KUKA KRL program: NEW_MASTER_MESA_A.src, NEW_MASTER_MESA_A.dat

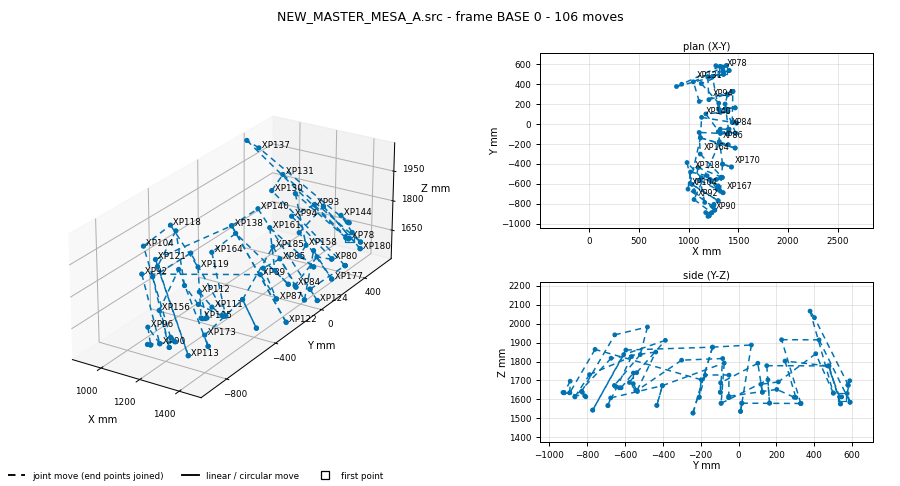
[picture p0: tool path of NEW_MASTER_MESA_A.src in frame BASE 0, 106 of 108 moves have a stored position in this frame; points joined in program order, loops and branches not executed]
--- NEW_MASTER_MESA_A.src ---
&ACCESS RVP
&REL 381
&PARAM EDITMASK = *
&PARAM TEMPLATE = C:\KRC\Roboter\Template\vorgabe
&PARAM DISKPATH = KRC:\R1\Program\Solda\MASTER_125
DEF NEW_MASTER_MESA_A( )
;FOLD INI;%{PE}
  ;FOLD BASISTECH INI
    GLOBAL INTERRUPT DECL 3 WHEN $STOPMESS==TRUE DO IR_STOPM ( )
    INTERRUPT ON 3
    BAS (#INITMOV,0 )
  ;ENDFOLD (BASISTECH INI)
  ;FOLD USER INI
    ;Make your modifications here

  ;ENDFOLD (USER INI)
;ENDFOLD (INI)

;FOLD PTP HOME  Vel= 100 % DEFAULT;%{PE}%MKUKATPBASIS,%CMOVE,%VPTP,%P 1:PTP, 2:HOME, 3:, 5:100, 7:DEFAULT
$BWDSTART = FALSE
PDAT_ACT=PDEFAULT
FDAT_ACT=FHOME
BAS (#PTP_PARAMS,100 )
$H_POS=XHOME
PTP  XHOME
;ENDFOLD
;FOLD ; CORDAO 01;%{PE}%R 8.3.48,%MKUKATPBASIS,%CCOMMENT,%VNORMAL,%P 2:CORDAO 01
;ENDFOLD
;FOLD ARCON WDAT39 PTP P78 Vel=100 % PDAT60 Tool[1]:TOCH Base[0] ;%{PE}
;FOLD Parameters ;%{h}
;Params IlfProvider=kukaroboter.arctech.arconptp; Kuka.PointName=P78; Kuka.BlendingEnabled=False; Kuka.MoveDataPtpName=PDAT60; Kuka.VelocityPtp=100; Kuka.MovementParameterFieldEnabled=True; ArcTech.WdatVarName=WDAT39; ArcTech.SeamName=
;ENDFOLD
$BWDSTART = FALSE
PDAT_ACT = PPDAT60
FDAT_ACT = FP78
BAS(#PTP_PARAMS, 100.0)
TRIGGER WHEN DISTANCE = 1 DELAY = ATBg_PreDefinitionTime DO Arc_DefineStrikeParams(3, AS_WDAT39) PRIO = -1
Arc_DefineCpPattern(#OffInAdvance, WV_WDAT39, TRUE)
PTP XP78
Arc_On(3, AS_WDAT39, ATBg_StartErrSetField[1], AW_WDAT39, WV_WDAT39, ATBg_WeldErrSetField[1], #StdArcOn, " ")
Arc_DefineCpPattern(#OnInAdvance, WV_WDAT39, TRUE)
;ENDFOLD
;FOLD ARCOFF WDAT40 LIN P79 CPDAT22 Tool[1]:TOCH Base[0] ;%{PE}
;FOLD Parameters ;%{h}
;Params IlfProvider=kukaroboter.arctech.arcofflin; Kuka.PointName=P79; Kuka.BlendingEnabled=False; Kuka.MoveDataName=CPDAT22;  Kuka.MovementParameterFieldEnabled=True; ArcTech.WdatVarName=WDAT40
;ENDFOLD
$BWDSTART = FALSE
LDAT_ACT = LCPDAT22
FDAT_ACT = FP79
BAS(#CP_PARAMS, ATBg_BAS_VELDefinition)
LIN XP79
Arc_Off(1, AC_WDAT40)
;ENDFOLD
;FOLD PTP P93 CONT Vel=100 % PDAT70 Tool[1]:TOCH Base[0];%{PE}%R 8.3.48,%MKUKATPBASIS,%CMOVE,%VPTP,%P 1:PTP, 2:P93, 3:C_DIS, 5:100, 7:PDAT70
$BWDSTART=FALSE
PDAT_ACT=PPDAT70
FDAT_ACT=FP93
BAS(#PTP_PARAMS,100)
PTP XP93 C_DIS
;ENDFOLD
;FOLD PTP P94 CONT Vel=100 % PDAT71 Tool[1]:TOCH Base[0];%{PE}%R 8.3.48,%MKUKATPBASIS,%CMOVE,%VPTP,%P 1:PTP, 2:P94, 3:C_DIS, 5:100, 7:PDAT71
$BWDSTART=FALSE
PDAT_ACT=PPDAT71
FDAT_ACT=FP94
BAS(#PTP_PARAMS,100)
PTP XP94 C_DIS
;ENDFOLD
;FOLD ; CORDAO 02;%{PE}%R 8.3.48,%MKUKATPBASIS,%CCOMMENT,%VNORMAL,%P 2:CORDAO 02
;ENDFOLD
;FOLD ARCON WDAT41 PTP P80 Vel=100 % PDAT61 Tool[1]:TOCH Base[0] ;%{PE}
;FOLD Parameters ;%{h}
;Params IlfProvider=kukaroboter.arctech.arconptp; Kuka.PointName=P80; Kuka.BlendingEnabled=False; Kuka.MoveDataPtpName=PDAT61; Kuka.VelocityPtp=100; Kuka.MovementParameterFieldEnabled=True; ArcTech.WdatVarName=WDAT41; ArcTech.SeamName=
;ENDFOLD
$BWDSTART = FALSE
PDAT_ACT = PPDAT61
FDAT_ACT = FP80
BAS(#PTP_PARAMS, 100.0)
TRIGGER WHEN DISTANCE = 1 DELAY = ATBg_PreDefinitionTime DO Arc_DefineStrikeParams(1, AS_WDAT41) PRIO = -1
Arc_DefineCpPattern(#OffInAdvance, WV_WDAT41, TRUE)
PTP XP80
Arc_On(1, AS_WDAT41, ATBg_StartErrSetField[1], AW_WDAT41, WV_WDAT41, ATBg_WeldErrSetField[1], #StdArcOn, " ")
Arc_DefineCpPattern(#OnInAdvance, WV_WDAT41, TRUE)
;ENDFOLD
;FOLD ARCOFF WDAT42 LIN P81 CPDAT23 Tool[1]:TOCH Base[0] ;%{PE}
;FOLD Parameters ;%{h}
;Params IlfProvider=kukaroboter.arctech.arcofflin; Kuka.PointName=P81; Kuka.BlendingEnabled=False; Kuka.MoveDataName=CPDAT23;  Kuka.MovementParameterFieldEnabled=True; ArcTech.WdatVarName=WDAT42
;ENDFOLD
$BWDSTART = FALSE
LDAT_ACT = LCPDAT23
FDAT_ACT = FP81
BAS(#CP_PARAMS, ATBg_BAS_VELDefinition)
LIN XP81
Arc_Off(1, AC_WDAT42)
;ENDFOLD
;FOLD PTP P95 CONT Vel=100 % PDAT72 Tool[1]:TOCH Base[0];%{PE}%R 8.3.48,%MKUKATPBASIS,%CMOVE,%VPTP,%P 1:PTP, 2:P95, 3:C_DIS, 5:100, 7:PDAT72
$BWDSTART=FALSE
PDAT_ACT=PPDAT72
FDAT_ACT=FP95
BAS(#PTP_PARAMS,100)
PTP XP95 C_DIS
;ENDFOLD
;FOLD PTP P84 CONT Vel=100 % PDAT63 Tool[1]:TOCH Base[0];%{PE}%R 8.3.48,%MKUKATPBASIS,%CMOVE,%VPTP,%P 1:PTP, 2:P84, 3:C_DIS, 5:100, 7:PDAT63
$BWDSTART=FALSE
PDAT_ACT=PPDAT63
FDAT_ACT=FP84
BAS(#PTP_PARAMS,100)
PTP XP84 C_DIS
;ENDFOLD
;FOLD ; CORDAO 03;%{PE}%R 8.3.48,%MKUKATPBASIS,%CCOMMENT,%VNORMAL,%P 2:CORDAO 03
;ENDFOLD
;FOLD ARCON WDAT43 PTP P82 Vel=100 % PDAT62 Tool[1]:TOCH Base[0] ;%{PE}
;FOLD Parameters ;%{h}
;Params IlfProvider=kukaroboter.arctech.arconptp; Kuka.PointName=P82; Kuka.BlendingEnabled=False; Kuka.MoveDataPtpName=PDAT62; Kuka.VelocityPtp=100; Kuka.MovementParameterFieldEnabled=True; ArcTech.WdatVarName=WDAT43; ArcTech.SeamName=
;ENDFOLD
$BWDSTART = FALSE
PDAT_ACT = PPDAT62
FDAT_ACT = FP82
BAS(#PTP_PARAMS, 100.0)
TRIGGER WHEN DISTANCE = 1 DELAY = ATBg_PreDefinitionTime DO Arc_DefineStrikeParams(1, AS_WDAT43) PRIO = -1
Arc_DefineCpPattern(#OffInAdvance, WV_WDAT43, TRUE)
PTP XP82
Arc_On(1, AS_WDAT43, ATBg_StartErrSetField[1], AW_WDAT43, WV_WDAT43, ATBg_WeldErrSetField[1], #StdArcOn, " ")
Arc_DefineCpPattern(#OnInAdvance, WV_WDAT43, TRUE)
;ENDFOLD
;FOLD ARCOFF WDAT44 LIN P83 CPDAT24 Tool[1]:TOCH Base[0] ;%{PE}
;FOLD Parameters ;%{h}
;Params IlfProvider=kukaroboter.arctech.arcofflin; Kuka.PointName=P83; Kuka.BlendingEnabled=False; Kuka.MoveDataName=CPDAT24;  Kuka.MovementParameterFieldEnabled=True; ArcTech.WdatVarName=WDAT44
;ENDFOLD
$BWDSTART = FALSE
LDAT_ACT = LCPDAT24
FDAT_ACT = FP83
BAS(#CP_PARAMS, ATBg_BAS_VELDefinition)
LIN XP83
Arc_Off(1, AC_WDAT44)
;ENDFOLD
;FOLD PTP P85 CONT Vel=100 % PDAT64 Tool[1]:TOCH Base[0];%{PE}%R 8.3.48,%MKUKATPBASIS,%CMOVE,%VPTP,%P 1:PTP, 2:P85, 3:C_DIS, 5:100, 7:PDAT64
$BWDSTART=FALSE
PDAT_ACT=PPDAT64
FDAT_ACT=FP85
BAS(#PTP_PARAMS,100)
PTP XP85 C_DIS
;ENDFOLD
;FOLD PTP P86 CONT Vel=100 % PDAT65 Tool[1]:TOCH Base[0];%{PE}%R 8.3.48,%MKUKATPBASIS,%CMOVE,%VPTP,%P 1:PTP, 2:P86, 3:C_DIS, 5:100, 7:PDAT65
$BWDSTART=FALSE
PDAT_ACT=PPDAT65
FDAT_ACT=FP86
BAS(#PTP_PARAMS,100)
PTP XP86 C_DIS
;ENDFOLD
;FOLD ; CORDAO 04;%{PE}%R 8.3.48,%MKUKATPBASIS,%CCOMMENT,%VNORMAL,%P 2:CORDAO 04
;ENDFOLD
;FOLD ARCON WDAT45 PTP P87 Vel=100 % PDAT66 Tool[1]:TOCH Base[0] ;%{PE}
;FOLD Parameters ;%{h}
;Params IlfProvider=kukaroboter.arctech.arconptp; Kuka.PointName=P87; Kuka.BlendingEnabled=False; Kuka.MoveDataPtpName=PDAT66; Kuka.VelocityPtp=100; Kuka.MovementParameterFieldEnabled=True; ArcTech.WdatVarName=WDAT45; ArcTech.SeamName=
;ENDFOLD
$BWDSTART = FALSE
PDAT_ACT = PPDAT66
FDAT_ACT = FP87
BAS(#PTP_PARAMS, 100.0)
TRIGGER WHEN DISTANCE = 1 DELAY = ATBg_PreDefinitionTime DO Arc_DefineStrikeParams(1, AS_WDAT45) PRIO = -1
Arc_DefineCpPattern(#OffInAdvance, WV_WDAT45, TRUE)
PTP XP87
Arc_On(1, AS_WDAT45, ATBg_StartErrSetField[1], AW_WDAT45, WV_WDAT45, ATBg_WeldErrSetField[1], #StdArcOn, " ")
Arc_DefineCpPattern(#OnInAdvance, WV_WDAT45, TRUE)
;ENDFOLD
;FOLD ARCOFF WDAT46 LIN P88 CPDAT25 Tool[1]:TOCH Base[0] ;%{PE}
;FOLD Parameters ;%{h}
;Params IlfProvider=kukaroboter.arctech.arcofflin; Kuka.PointName=P88; Kuka.BlendingEnabled=False; Kuka.MoveDataName=CPDAT25;  Kuka.MovementParameterFieldEnabled=True; ArcTech.WdatVarName=WDAT46
;ENDFOLD
$BWDSTART = FALSE
LDAT_ACT = LCPDAT25
FDAT_ACT = FP88
BAS(#CP_PARAMS, ATBg_BAS_VELDefinition)
LIN XP88
Arc_Off(1, AC_WDAT46)
;ENDFOLD
;FOLD PTP P89 CONT Vel=100 % PDAT67 Tool[1]:TOCH Base[0];%{PE}%R 8.3.48,%MKUKATPBASIS,%CMOVE,%VPTP,%P 1:PTP, 2:P89, 3:C_DIS, 5:100, 7:PDAT67
$BWDSTART=FALSE
PDAT_ACT=PPDAT67
FDAT_ACT=FP89
BAS(#PTP_PARAMS,100)
PTP XP89 C_DIS
;ENDFOLD
;FOLD PTP P92 CONT Vel=100 % PDAT69 Tool[1]:TOCH Base[0];%{PE}%R 8.3.48,%MKUKATPBASIS,%CMOVE,%VPTP,%P 1:PTP, 2:P92, 3:C_DIS, 5:100, 7:PDAT69
$BWDSTART=FALSE
PDAT_ACT=PPDAT69
FDAT_ACT=FP92
BAS(#PTP_PARAMS,100)
PTP XP92 C_DIS
;ENDFOLD
;FOLD ; CORDAO 05;%{PE}%R 8.3.48,%MKUKATPBASIS,%CCOMMENT,%VNORMAL,%P 2:CORDAO 05
;ENDFOLD
;FOLD ARCON WDAT47 PTP P90 Vel=100 % PDAT68 Tool[1]:TOCH Base[0] ;%{PE}
;FOLD Parameters ;%{h}
;Params IlfProvider=kukaroboter.arctech.arconptp; Kuka.PointName=P90; Kuka.BlendingEnabled=False; Kuka.MoveDataPtpName=PDAT68; Kuka.VelocityPtp=100; Kuka.MovementParameterFieldEnabled=True; ArcTech.WdatVarName=WDAT47; ArcTech.SeamName=
;ENDFOLD
$BWDSTART = FALSE
PDAT_ACT = PPDAT68
FDAT_ACT = FP90
BAS(#PTP_PARAMS, 100.0)
TRIGGER WHEN DISTANCE = 1 DELAY = ATBg_PreDefinitionTime DO Arc_DefineStrikeParams(1, AS_WDAT47) PRIO = -1
Arc_DefineCpPattern(#OffInAdvance, WV_WDAT47, TRUE)
PTP XP90
Arc_On(1, AS_WDAT47, ATBg_StartErrSetField[1], AW_WDAT47, WV_WDAT47, ATBg_WeldErrSetField[1], #StdArcOn, " ")
Arc_DefineCpPattern(#OnInAdvance, WV_WDAT47, TRUE)
;ENDFOLD
;FOLD ARCOFF WDAT48 LIN P91 CPDAT26 Tool[1]:TOCH Base[0] ;%{PE}
;FOLD Parameters ;%{h}
;Params IlfProvider=kukaroboter.arctech.arcofflin; Kuka.PointName=P91; Kuka.BlendingEnabled=False; Kuka.MoveDataName=CPDAT26;  Kuka.MovementParameterFieldEnabled=True; ArcTech.WdatVarName=WDAT48
;ENDFOLD
$BWDSTART = FALSE
LDAT_ACT = LCPDAT26
FDAT_ACT = FP91
BAS(#CP_PARAMS, ATBg_BAS_VELDefinition)
LIN XP91
Arc_Off(1, AC_WDAT48)
;ENDFOLD
;FOLD PTP P96 CONT Vel=100 % PDAT73 Tool[1]:TOCH Base[0];%{PE}%R 8.3.48,%MKUKATPBASIS,%CMOVE,%VPTP,%P 1:PTP, 2:P96, 3:C_DIS, 5:100, 7:PDAT73
$BWDSTART=FALSE
PDAT_ACT=PPDAT73
FDAT_ACT=FP96
BAS(#PTP_PARAMS,100)
PTP XP96 C_DIS
;ENDFOLD
;FOLD ; CORDAO 06;%{PE}%R 8.3.48,%MKUKATPBASIS,%CCOMMENT,%VNORMAL,%P 2:CORDAO 06
;ENDFOLD
;FOLD ARCON WDAT49 PTP P97 Vel=100 % PDAT74 Tool[1]:TOCH Base[0] ;%{PE}
;FOLD Parameters ;%{h}
;Params IlfProvider=kukaroboter.arctech.arconptp; Kuka.PointName=P97; Kuka.BlendingEnabled=False; Kuka.MoveDataPtpName=PDAT74; Kuka.VelocityPtp=100; Kuka.MovementParameterFieldEnabled=True; ArcTech.WdatVarName=WDAT49; ArcTech.SeamName=
;ENDFOLD
$BWDSTART = FALSE
PDAT_ACT = PPDAT74
FDAT_ACT = FP97
BAS(#PTP_PARAMS, 100.0)
TRIGGER WHEN DISTANCE = 1 DELAY = ATBg_PreDefinitionTime DO Arc_DefineStrikeParams(1, AS_WDAT49) PRIO = -1
Arc_DefineCpPattern(#OffInAdvance, WV_WDAT49, TRUE)
PTP XP97
Arc_On(1, AS_WDAT49, ATBg_StartErrSetField[1], AW_WDAT49, WV_WDAT49, ATBg_WeldErrSetField[1], #StdArcOn, " ")
Arc_DefineCpPattern(#OnInAdvance, WV_WDAT49, TRUE)
;ENDFOLD
;FOLD ARCOFF WDAT50 LIN P98 CPDAT27 Tool[1]:TOCH Base[0] ;%{PE}
;FOLD Parameters ;%{h}
;Params IlfProvider=kukaroboter.arctech.arcofflin; Kuka.PointName=P98; Kuka.BlendingEnabled=False; Kuka.MoveDataName=CPDAT27;  Kuka.MovementParameterFieldEnabled=True; ArcTech.WdatVarName=WDAT50
;ENDFOLD
$BWDSTART = FALSE
LDAT_ACT = LCPDAT27
FDAT_ACT = FP98
BAS(#CP_PARAMS, ATBg_BAS_VELDefinition)
LIN XP98
Arc_Off(1, AC_WDAT50)
;ENDFOLD
;FOLD ARCOFF WDAT51 LIN P99 CPDAT28 Tool[1]:TOCH Base[0] ;%{PE}
;FOLD Parameters ;%{h}
;Params IlfProvider=kukaroboter.arctech.arcofflin; Kuka.PointName=P99; Kuka.BlendingEnabled=False; Kuka.MoveDataName=CPDAT28;  Kuka.MovementParameterFieldEnabled=True; ArcTech.WdatVarName=WDAT51
;ENDFOLD
$BWDSTART = FALSE
LDAT_ACT = LCPDAT28
FDAT_ACT = FP99
BAS(#CP_PARAMS, ATBg_BAS_VELDefinition)
LIN XP99
Arc_Off(1, AC_WDAT51)
;ENDFOLD
;FOLD ; CORDAO 07;%{PE}%R 8.3.48,%MKUKATPBASIS,%CCOMMENT,%VNORMAL,%P 2:CORDAO 07
;ENDFOLD
;FOLD ARCON WDAT52 PTP P100 Vel=100 % PDAT75 Tool[1]:TOCH Base[0] ;%{PE}
;FOLD Parameters ;%{h}
;Params IlfProvider=kukaroboter.arctech.arconptp; Kuka.PointName=P100; Kuka.BlendingEnabled=False; Kuka.MoveDataPtpName=PDAT75; Kuka.VelocityPtp=100; Kuka.MovementParameterFieldEnabled=True; ArcTech.WdatVarName=WDAT52; ArcTech.SeamName=
;ENDFOLD
$BWDSTART = FALSE
PDAT_ACT = PPDAT75
FDAT_ACT = FP100
BAS(#PTP_PARAMS, 100.0)
TRIGGER WHEN DISTANCE = 1 DELAY = ATBg_PreDefinitionTime DO Arc_DefineStrikeParams(1, AS_WDAT52) PRIO = -1
Arc_DefineCpPattern(#OffInAdvance, WV_WDAT52, TRUE)
PTP XP100
Arc_On(1, AS_WDAT52, ATBg_StartErrSetField[1], AW_WDAT52, WV_WDAT52, ATBg_WeldErrSetField[1], #StdArcOn, " ")
Arc_DefineCpPattern(#OnInAdvance, WV_WDAT52, TRUE)
;ENDFOLD
;FOLD ARCOFF WDAT53 LIN P101 CPDAT29 Tool[1]:TOCH Base[0] ;%{PE}
;FOLD Parameters ;%{h}
;Params IlfProvider=kukaroboter.arctech.arcofflin; Kuka.PointName=P101; Kuka.BlendingEnabled=False; Kuka.MoveDataName=CPDAT29;  Kuka.MovementParameterFieldEnabled=True; ArcTech.WdatVarName=WDAT53
;ENDFOLD
$BWDSTART = FALSE
LDAT_ACT = LCPDAT29
FDAT_ACT = FP101
BAS(#CP_PARAMS, ATBg_BAS_VELDefinition)
LIN XP101
Arc_Off(1, AC_WDAT53)
;ENDFOLD
;FOLD ; CORDAO 08;%{PE}%R 8.3.48,%MKUKATPBASIS,%CCOMMENT,%VNORMAL,%P 2:CORDAO 08
;ENDFOLD
;FOLD ARCON WDAT54 PTP P102 Vel=100 % PDAT76 Tool[1]:TOCH Base[0] ;%{PE}
;FOLD Parameters ;%{h}
;Params IlfProvider=kukaroboter.arctech.arconptp; Kuka.PointName=P102; Kuka.BlendingEnabled=False; Kuka.MoveDataPtpName=PDAT76; Kuka.VelocityPtp=100; Kuka.MovementParameterFieldEnabled=True; ArcTech.WdatVarName=WDAT54; ArcTech.SeamName=
;ENDFOLD
$BWDSTART = FALSE
PDAT_ACT = PPDAT76
FDAT_ACT = FP102
BAS(#PTP_PARAMS, 100.0)
TRIGGER WHEN DISTANCE = 1 DELAY = ATBg_PreDefinitionTime DO Arc_DefineStrikeParams(1, AS_WDAT54) PRIO = -1
Arc_DefineCpPattern(#OffInAdvance, WV_WDAT54, TRUE)
PTP XP102
Arc_On(1, AS_WDAT54, ATBg_StartErrSetField[1], AW_WDAT54, WV_WDAT54, ATBg_WeldErrSetField[1], #StdArcOn, " ")
Arc_DefineCpPattern(#OnInAdvance, WV_WDAT54, TRUE)
;ENDFOLD
;FOLD ARCOFF WDAT55 LIN P103 CPDAT30 Tool[1]:TOCH Base[0] ;%{PE}
;FOLD Parameters ;%{h}
;Params IlfProvider=kukaroboter.arctech.arcofflin; Kuka.PointName=P103; Kuka.BlendingEnabled=False; Kuka.MoveDataName=CPDAT30;  Kuka.MovementParameterFieldEnabled=True; ArcTech.WdatVarName=WDAT55
;ENDFOLD
$BWDSTART = FALSE
LDAT_ACT = LCPDAT30
FDAT_ACT = FP103
BAS(#CP_PARAMS, ATBg_BAS_VELDefinition)
LIN XP103
Arc_Off(1, AC_WDAT55)
;ENDFOLD
;FOLD PTP P104 CONT Vel=100 % PDAT77 Tool[1]:TOCH Base[0];%{PE}%R 8.3.48,%MKUKATPBASIS,%CMOVE,%VPTP,%P 1:PTP, 2:P104, 3:C_DIS, 5:100, 7:PDAT77
$BWDSTART=FALSE
PDAT_ACT=PPDAT77
FDAT_ACT=FP104
BAS(#PTP_PARAMS,100)
PTP XP104 C_DIS
;ENDFOLD
;FOLD PTP P118 CONT Vel=100 % PDAT88 Tool[1]:TOCH Base[0];%{PE}%R 8.3.48,%MKUKATPBASIS,%CMOVE,%VPTP,%P 1:PTP, 2:P118, 3:C_DIS, 5:100, 7:PDAT88
$BWDSTART=FALSE
PDAT_ACT=PPDAT88
FDAT_ACT=FP118
BAS(#PTP_PARAMS,100)
PTP XP118 C_DIS
;ENDFOLD
;FOLD PTP P119 CONT Vel=100 % PDAT89 Tool[1]:TOCH Base[0];%{PE}%R 8.3.48,%MKUKATPBASIS,%CMOVE,%VPTP,%P 1:PTP, 2:P119, 3:C_DIS, 5:100, 7:PDAT89
$BWDSTART=FALSE
PDAT_ACT=PPDAT89
FDAT_ACT=FP119
BAS(#PTP_PARAMS,100)
PTP XP119 C_DIS
;ENDFOLD
;FOLD ; CORDAO 09;%{PE}%R 8.3.48,%MKUKATPBASIS,%CCOMMENT,%VNORMAL,%P 2:CORDAO 09
;ENDFOLD
;FOLD ARCON WDAT56 PTP P105 Vel=100 % PDAT78 Tool[1]:TOCH Base[0] ;%{PE}
;FOLD Parameters ;%{h}
;Params IlfProvider=kukaroboter.arctech.arconptp; Kuka.PointName=P105; Kuka.BlendingEnabled=False; Kuka.MoveDataPtpName=PDAT78; Kuka.VelocityPtp=100; Kuka.MovementParameterFieldEnabled=True; ArcTech.WdatVarName=WDAT56; ArcTech.SeamName=
;ENDFOLD
$BWDSTART = FALSE
PDAT_ACT = PPDAT78
FDAT_ACT = FP105
BAS(#PTP_PARAMS, 100.0)
TRIGGER WHEN DISTANCE = 1 DELAY = ATBg_PreDefinitionTime DO Arc_DefineStrikeParams(1, AS_WDAT56) PRIO = -1
Arc_DefineCpPattern(#OffInAdvance, WV_WDAT56, TRUE)
PTP XP105
Arc_On(1, AS_WDAT56, ATBg_StartErrSetField[1], AW_WDAT56, WV_WDAT56, ATBg_WeldErrSetField[1], #StdArcOn, " ")
Arc_DefineCpPattern(#OnInAdvance, WV_WDAT56, TRUE)
;ENDFOLD
;FOLD ARCOFF WDAT57 LIN P106 CPDAT31 Tool[1]:TOCH Base[0] ;%{PE}
;FOLD Parameters ;%{h}
;Params IlfProvider=kukaroboter.arctech.arcofflin; Kuka.PointName=P106; Kuka.BlendingEnabled=False; Kuka.MoveDataName=CPDAT31;  Kuka.MovementParameterFieldEnabled=True; ArcTech.WdatVarName=WDAT57
;ENDFOLD
$BWDSTART = FALSE
LDAT_ACT = LCPDAT31
FDAT_ACT = FP106
BAS(#CP_PARAMS, ATBg_BAS_VELDefinition)
LIN XP106
Arc_Off(1, AC_WDAT57)
;ENDFOLD
;FOLD ; CORDAO 10;%{PE}%R 8.3.48,%MKUKATPBASIS,%CCOMMENT,%VNORMAL,%P 2:CORDAO 10
;ENDFOLD
;FOLD ARCON WDAT58 PTP P107 Vel=100 % PDAT79 Tool[1]:TOCH Base[0] ;%{PE}
;FOLD Parameters ;%{h}
;Params IlfProvider=kukaroboter.arctech.arconptp; Kuka.PointName=P107; Kuka.BlendingEnabled=False; Kuka.MoveDataPtpName=PDAT79; Kuka.VelocityPtp=100; Kuka.MovementParameterFieldEnabled=True; ArcTech.WdatVarName=WDAT58; ArcTech.SeamName=
;ENDFOLD
$BWDSTART = FALSE
PDAT_ACT = PPDAT79
FDAT_ACT = FP107
BAS(#PTP_PARAMS, 100.0)
TRIGGER WHEN DISTANCE = 1 DELAY = ATBg_PreDefinitionTime DO Arc_DefineStrikeParams(1, AS_WDAT58) PRIO = -1
Arc_DefineCpPattern(#OffInAdvance, WV_WDAT58, TRUE)
PTP XP107
Arc_On(1, AS_WDAT58, ATBg_StartErrSetField[1], AW_WDAT58, WV_WDAT58, ATBg_WeldErrSetField[1], #StdArcOn, " ")
Arc_DefineCpPattern(#OnInAdvance, WV_WDAT58, TRUE)
;ENDFOLD
;FOLD ARCOFF WDAT59 LIN P108 CPDAT32 Tool[1]:TOCH Base[0] ;%{PE}
;FOLD Parameters ;%{h}
;Params IlfProvider=kukaroboter.arctech.arcofflin; Kuka.PointName=P108; Kuka.BlendingEnabled=False; Kuka.MoveDataName=CPDAT32;  Kuka.MovementParameterFieldEnabled=True; ArcTech.WdatVarName=WDAT59
;ENDFOLD
$BWDSTART = FALSE
LDAT_ACT = LCPDAT32
FDAT_ACT = FP108
BAS(#CP_PARAMS, ATBg_BAS_VELDefinition)
LIN XP108
Arc_Off(1, AC_WDAT59)
;ENDFOLD
;FOLD PTP P112 CONT Vel=100 % PDAT82 Tool[1]:TOCH Base[0];%{PE}%R 8.3.48,%MKUKATPBASIS,%CMOVE,%VPTP,%P 1:PTP, 2:P112, 3:C_DIS, 5:100, 7:PDAT82
$BWDSTART=FALSE
PDAT_ACT=PPDAT82
FDAT_ACT=FP112
BAS(#PTP_PARAMS,100)
PTP XP112 C_DIS
;ENDFOLD
;FOLD PTP P111 CONT Vel=100 % PDAT81 Tool[1]:TOCH Base[0];%{PE}%R 8.3.48,%MKUKATPBASIS,%CMOVE,%VPTP,%P 1:PTP, 2:P111, 3:C_DIS, 5:100, 7:PDAT81
$BWDSTART=FALSE
PDAT_ACT=PPDAT81
FDAT_ACT=FP111
BAS(#PTP_PARAMS,100)
PTP XP111 C_DIS
;ENDFOLD
;FOLD ; CORDAO 11;%{PE}%R 8.3.48,%MKUKATPBASIS,%CCOMMENT,%VNORMAL,%P 2:CORDAO 11
;ENDFOLD
;FOLD ARCON WDAT60 PTP P109 Vel=100 % PDAT80 Tool[1]:TOCH Base[0] ;%{PE}
;FOLD Parameters ;%{h}
;Params IlfProvider=kukaroboter.arctech.arconptp; Kuka.PointName=P109; Kuka.BlendingEnabled=False; Kuka.MoveDataPtpName=PDAT80; Kuka.VelocityPtp=100; Kuka.MovementParameterFieldEnabled=True; ArcTech.WdatVarName=WDAT60; ArcTech.SeamName=
;ENDFOLD
$BWDSTART = FALSE
PDAT_ACT = PPDAT80
FDAT_ACT = FP109
BAS(#PTP_PARAMS, 100.0)
TRIGGER WHEN DISTANCE = 1 DELAY = ATBg_PreDefinitionTime DO Arc_DefineStrikeParams(1, AS_WDAT60) PRIO = -1
Arc_DefineCpPattern(#OffInAdvance, WV_WDAT60, TRUE)
PTP XP109
Arc_On(1, AS_WDAT60, ATBg_StartErrSetField[1], AW_WDAT60, WV_WDAT60, ATBg_WeldErrSetField[1], #StdArcOn, " ")
Arc_DefineCpPattern(#OnInAdvance, WV_WDAT60, TRUE)
;ENDFOLD
;FOLD ARCOFF WDAT61 LIN P110 CPDAT33 Tool[1]:TOCH Base[0] ;%{PE}
;FOLD Parameters ;%{h}
;Params IlfProvider=kukaroboter.arctech.arcofflin; Kuka.PointName=P110; Kuka.BlendingEnabled=False; Kuka.MoveDataName=CPDAT33;  Kuka.MovementParameterFieldEnabled=True; ArcTech.WdatVarName=WDAT61
;ENDFOLD
$BWDSTART = FALSE
LDAT_ACT = LCPDAT33
FDAT_ACT = FP110
BAS(#CP_PARAMS, ATBg_BAS_VELDefinition)
LIN XP110
Arc_Off(1, AC_WDAT61)
;ENDFOLD
;FOLD PTP P117 CONT Vel=100 % PDAT87 Tool[1]:TOCH Base[0];%{PE}%R 8.3.48,%MKUKATPBASIS,%CMOVE,%VPTP,%P 1:PTP, 2:P117, 3:C_DIS, 5:100, 7:PDAT87
$BWDSTART=FALSE
PDAT_ACT=PPDAT87
FDAT_ACT=FP117
BAS(#PTP_PARAMS,100)
PTP XP117 C_DIS
;ENDFOLD
;FOLD PTP P116 CONT Vel=100 % PDAT86 Tool[1]:TOCH Base[0];%{PE}%R 8.3.48,%MKUKATPBASIS,%CMOVE,%VPTP,%P 1:PTP, 2:P116, 3:C_DIS, 5:100, 7:PDAT86
$BWDSTART=FALSE
PDAT_ACT=PPDAT86
FDAT_ACT=FP116
BAS(#PTP_PARAMS,100)
PTP XP116 C_DIS
;ENDFOLD
;FOLD PTP P115 CONT Vel=100 % PDAT85 Tool[1]:TOCH Base[0];%{PE}%R 8.3.48,%MKUKATPBASIS,%CMOVE,%VPTP,%P 1:PTP, 2:P115, 3:C_DIS, 5:100, 7:PDAT85
$BWDSTART=FALSE
PDAT_ACT=PPDAT85
FDAT_ACT=FP115
BAS(#PTP_PARAMS,100)
PTP XP115 C_DIS
;ENDFOLD
;FOLD PTP P114 CONT Vel=100 % PDAT84 Tool[1]:TOCH Base[0];%{PE}%R 8.3.48,%MKUKATPBASIS,%CMOVE,%VPTP,%P 1:PTP, 2:P114, 3:C_DIS, 5:100, 7:PDAT84
$BWDSTART=FALSE
PDAT_ACT=PPDAT84
FDAT_ACT=FP114
BAS(#PTP_PARAMS,100)
PTP XP114 C_DIS
;ENDFOLD
;FOLD ; CORDAO 12;%{PE}%R 8.3.48,%MKUKATPBASIS,%CCOMMENT,%VNORMAL,%P 2:CORDAO 12
;ENDFOLD
;FOLD ARCON WDAT62 PTP P113 Vel=100 % PDAT83 Tool[1]:TOCH Base[0] ;%{PE}
;FOLD Parameters ;%{h}
;Params IlfProvider=kukaroboter.arctech.arconptp; Kuka.PointName=P113; Kuka.BlendingEnabled=False; Kuka.MoveDataPtpName=PDAT83; Kuka.VelocityPtp=100; Kuka.MovementParameterFieldEnabled=True; ArcTech.WdatVarName=WDAT62; ArcTech.SeamName=
;ENDFOLD
$BWDSTART = FALSE
PDAT_ACT = PPDAT83
FDAT_ACT = FP113
BAS(#PTP_PARAMS, 100.0)
TRIGGER WHEN DISTANCE = 1 DELAY = ATBg_PreDefinitionTime DO Arc_DefineStrikeParams(1, AS_WDAT62) PRIO = -1
Arc_DefineCpPattern(#OffInAdvance, WV_WDAT62, TRUE)
PTP XP113
Arc_On(1, AS_WDAT62, ATBg_StartErrSetField[1], AW_WDAT62, WV_WDAT62, ATBg_WeldErrSetField[1], #StdArcOn, " ")
Arc_DefineCpPattern(#OnInAdvance, WV_WDAT62, TRUE)
;ENDFOLD
;FOLD ARCOFF WDAT63 LIN P120 CPDAT34 Tool[1]:TOCH Base[0] ;%{PE}
;FOLD Parameters ;%{h}
;Params IlfProvider=kukaroboter.arctech.arcofflin; Kuka.PointName=P120; Kuka.BlendingEnabled=False; Kuka.MoveDataName=CPDAT34;  Kuka.MovementParameterFieldEnabled=True; ArcTech.WdatVarName=WDAT63
;ENDFOLD
$BWDSTART = FALSE
LDAT_ACT = LCPDAT34
FDAT_ACT = FP120
BAS(#CP_PARAMS, ATBg_BAS_VELDefinition)
LIN XP120
Arc_Off(1, AC_WDAT63)
;ENDFOLD
;FOLD PTP P121 CONT Vel=100 % PDAT90 Tool[1]:TOCH Base[0];%{PE}%R 8.3.48,%MKUKATPBASIS,%CMOVE,%VPTP,%P 1:PTP, 2:P121, 3:C_DIS, 5:100, 7:PDAT90
$BWDSTART=FALSE
PDAT_ACT=PPDAT90
FDAT_ACT=FP121
BAS(#PTP_PARAMS,100)
PTP XP121 C_DIS
;ENDFOLD
;FOLD PTP P138 CONT Vel=100 % PDAT101 Tool[1]:TOCH Base[0];%{PE}%R 8.3.48,%MKUKATPBASIS,%CMOVE,%VPTP,%P 1:PTP, 2:P138, 3:C_DIS, 5:100, 7:PDAT101
$BWDSTART=FALSE
PDAT_ACT=PPDAT101
FDAT_ACT=FP138
BAS(#PTP_PARAMS,100)
PTP XP138 C_DIS
;ENDFOLD
;FOLD ; CORDAO 13;%{PE}%R 8.3.48,%MKUKATPBASIS,%CCOMMENT,%VNORMAL,%P 2:CORDAO 13
;ENDFOLD
;FOLD ARCON WDAT64 PTP P122 Vel=100 % PDAT91 Tool[1]:TOCH Base[0] ;%{PE}
;FOLD Parameters ;%{h}
;Params IlfProvider=kukaroboter.arctech.arconptp; Kuka.PointName=P122; Kuka.BlendingEnabled=False; Kuka.MoveDataPtpName=PDAT91; Kuka.VelocityPtp=100; Kuka.MovementParameterFieldEnabled=True; ArcTech.WdatVarName=WDAT64; ArcTech.SeamName=
;ENDFOLD
$BWDSTART = FALSE
PDAT_ACT = PPDAT91
FDAT_ACT = FP122
BAS(#PTP_PARAMS, 100.0)
TRIGGER WHEN DISTANCE = 1 DELAY = ATBg_PreDefinitionTime DO Arc_DefineStrikeParams(1, AS_WDAT64) PRIO = -1
Arc_DefineCpPattern(#OffInAdvance, WV_WDAT64, TRUE)
PTP XP122
Arc_On(1, AS_WDAT64, ATBg_StartErrSetField[1], AW_WDAT64, WV_WDAT64, ATBg_WeldErrSetField[1], #StdArcOn, " ")
Arc_DefineCpPattern(#OnInAdvance, WV_WDAT64, TRUE)
;ENDFOLD
;FOLD ARCOFF WDAT65 LIN P123 CPDAT35 Tool[1]:TOCH Base[0] ;%{PE}
;FOLD Parameters ;%{h}
;Params IlfProvider=kukaroboter.arctech.arcofflin; Kuka.PointName=P123; Kuka.BlendingEnabled=False; Kuka.MoveDataName=CPDAT35;  Kuka.MovementParameterFieldEnabled=True; ArcTech.WdatVarName=WDAT65
;ENDFOLD
$BWDSTART = FALSE
LDAT_ACT = LCPDAT35
FDAT_ACT = FP123
BAS(#CP_PARAMS, ATBg_BAS_VELDefinition)
LIN XP123
Arc_Off(1, AC_WDAT65)
;ENDFOLD
;FOLD PTP P139 CONT Vel=100 % PDAT102 Tool[1]:TOCH Base[0];%{PE}%R 8.3.48,%MKUKATPBASIS,%CMOVE,%VPTP,%P 1:PTP, 2:P139, 3:C_DIS, 5:100, 7:PDAT102
$BWDSTART=FALSE
PDAT_ACT=PPDAT102
FDAT_ACT=FP139
BAS(#PTP_PARAMS,100)
PTP XP139 C_DIS
;ENDFOLD
;FOLD PTP P140 CONT Vel=100 % PDAT103 Tool[1]:TOCH Base[0];%{PE}%R 8.3.48,%MKUKATPBASIS,%CMOVE,%VPTP,%P 1:PTP, 2:P140, 3:C_DIS, 5:100, 7:PDAT103
$BWDSTART=FALSE
PDAT_ACT=PPDAT103
FDAT_ACT=FP140
BAS(#PTP_PARAMS,100)
PTP XP140 C_DIS
;ENDFOLD
;FOLD PTP P141 CONT Vel=100 % PDAT104 Tool[1]:TOCH Base[0];%{PE}%R 8.3.48,%MKUKATPBASIS,%CMOVE,%VPTP,%P 1:PTP, 2:P141, 3:C_DIS, 5:100, 7:PDAT104
$BWDSTART=FALSE
PDAT_ACT=PPDAT104
FDAT_ACT=FP141
BAS(#PTP_PARAMS,100)
PTP XP141 C_DIS
;ENDFOLD
;FOLD ; CORDAO 14;%{PE}%R 8.3.48,%MKUKATPBASIS,%CCOMMENT,%VNORMAL,%P 2:CORDAO 14
;ENDFOLD
;FOLD ARCON WDAT66 PTP P124 Vel=100 % PDAT92 Tool[1]:TOCH Base[0] ;%{PE}
;FOLD Parameters ;%{h}
;Params IlfProvider=kukaroboter.arctech.arconptp; Kuka.PointName=P124; Kuka.BlendingEnabled=False; Kuka.MoveDataPtpName=PDAT92; Kuka.VelocityPtp=100; Kuka.MovementParameterFieldEnabled=True; ArcTech.WdatVarName=WDAT66; ArcTech.SeamName=
;ENDFOLD
$BWDSTART = FALSE
PDAT_ACT = PPDAT92
FDAT_ACT = FP124
BAS(#PTP_PARAMS, 100.0)
TRIGGER WHEN DISTANCE = 1 DELAY = ATBg_PreDefinitionTime DO Arc_DefineStrikeParams(1, AS_WDAT66) PRIO = -1
Arc_DefineCpPattern(#OffInAdvance, WV_WDAT66, TRUE)
PTP XP124
Arc_On(1, AS_WDAT66, ATBg_StartErrSetField[1], AW_WDAT66, WV_WDAT66, ATBg_WeldErrSetField[1], #StdArcOn, " ")
Arc_DefineCpPattern(#OnInAdvance, WV_WDAT66, TRUE)
;ENDFOLD
;FOLD ARCOFF WDAT67 LIN P125 CPDAT36 Tool[1]:TOCH Base[0] ;%{PE}
;FOLD Parameters ;%{h}
;Params IlfProvider=kukaroboter.arctech.arcofflin; Kuka.PointName=P125; Kuka.BlendingEnabled=False; Kuka.MoveDataName=CPDAT36;  Kuka.MovementParameterFieldEnabled=True; ArcTech.WdatVarName=WDAT67
;ENDFOLD
$BWDSTART = FALSE
LDAT_ACT = LCPDAT36
FDAT_ACT = FP125
BAS(#CP_PARAMS, ATBg_BAS_VELDefinition)
LIN XP125
Arc_Off(1, AC_WDAT67)
;ENDFOLD
;FOLD PTP P142 CONT Vel=100 % PDAT105 Tool[1]:TOCH Base[0];%{PE}%R 8.3.48,%MKUKATPBASIS,%CMOVE,%VPTP,%P 1:PTP, 2:P142, 3:C_DIS, 5:100, 7:PDAT105
$BWDSTART=FALSE
PDAT_ACT=PPDAT105
FDAT_ACT=FP142
BAS(#PTP_PARAMS,100)
PTP XP142 C_DIS
;ENDFOLD
;FOLD ; CORDAO 15;%{PE}%R 8.3.48,%MKUKATPBASIS,%CCOMMENT,%VNORMAL,%P 2:CORDAO 15
;ENDFOLD
;FOLD ARCON WDAT68 PTP P126 Vel=100 % PDAT93 Tool[1]:TOCH Base[0] ;%{PE}
;FOLD Parameters ;%{h}
;Params IlfProvider=kukaroboter.arctech.arconptp; Kuka.PointName=P126; Kuka.BlendingEnabled=False; Kuka.MoveDataPtpName=PDAT93; Kuka.VelocityPtp=100; Kuka.MovementParameterFieldEnabled=True; ArcTech.WdatVarName=WDAT68; ArcTech.SeamName=
;ENDFOLD
$BWDSTART = FALSE
PDAT_ACT = PPDAT93
FDAT_ACT = FP126
BAS(#PTP_PARAMS, 100.0)
TRIGGER WHEN DISTANCE = 1 DELAY = ATBg_PreDefinitionTime DO Arc_DefineStrikeParams(1, AS_WDAT68) PRIO = -1
Arc_DefineCpPattern(#OffInAdvance, WV_WDAT68, TRUE)
PTP XP126
Arc_On(1, AS_WDAT68, ATBg_StartErrSetField[1], AW_WDAT68, WV_WDAT68, ATBg_WeldErrSetField[1], #StdArcOn, " ")
Arc_DefineCpPattern(#OnInAdvance, WV_WDAT68, TRUE)
;ENDFOLD
;FOLD ARCOFF WDAT69 LIN P127 CPDAT37 Tool[1]:TOCH Base[0] ;%{PE}
;FOLD Parameters ;%{h}
;Params IlfProvider=kukaroboter.arctech.arcofflin; Kuka.PointName=P127; Kuka.BlendingEnabled=False; Kuka.MoveDataName=CPDAT37;  Kuka.MovementParameterFieldEnabled=True; ArcTech.WdatVarName=WDAT69
;ENDFOLD
$BWDSTART = FALSE
LDAT_ACT = LCPDAT37
FDAT_ACT = FP127
BAS(#CP_PARAMS, ATBg_BAS_VELDefinition)
LIN XP127
Arc_Off(1, AC_WDAT69)
;ENDFOLD
;FOLD ; CORDAO 16;%{PE}%R 8.3.48,%MKUKATPBASIS,%CCOMMENT,%VNORMAL,%P 2:CORDAO 16
;ENDFOLD
;FOLD ARCON WDAT70 PTP P128 Vel=100 % PDAT94 Tool[1]:TOCH Base[0] ;%{PE}
;FOLD Parameters ;%{h}
;Params IlfProvider=kukaroboter.arctech.arconptp; Kuka.PointName=P128; Kuka.BlendingEnabled=False; Kuka.MoveDataPtpName=PDAT94; Kuka.VelocityPtp=100; Kuka.MovementParameterFieldEnabled=True; ArcTech.WdatVarName=WDAT70; ArcTech.SeamName=
;ENDFOLD
$BWDSTART = FALSE
PDAT_ACT = PPDAT94
FDAT_ACT = FP128
BAS(#PTP_PARAMS, 100.0)
TRIGGER WHEN DISTANCE = 1 DELAY = ATBg_PreDefinitionTime DO Arc_DefineStrikeParams(1, AS_WDAT70) PRIO = -1
Arc_DefineCpPattern(#OffInAdvance, WV_WDAT70, TRUE)
PTP XP128
Arc_On(1, AS_WDAT70, ATBg_StartErrSetField[1], AW_WDAT70, WV_WDAT70, ATBg_WeldErrSetField[1], #StdArcOn, " ")
Arc_DefineCpPattern(#OnInAdvance, WV_WDAT70, TRUE)
;ENDFOLD
;FOLD ARCOFF WDAT71 LIN P129 CPDAT38 Tool[1]:TOCH Base[0] ;%{PE}
;FOLD Parameters ;%{h}
;Params IlfProvider=kukaroboter.arctech.arcofflin; Kuka.PointName=P129; Kuka.BlendingEnabled=False; Kuka.MoveDataName=CPDAT38;  Kuka.MovementParameterFieldEnabled=True; ArcTech.WdatVarName=WDAT71
;ENDFOLD
$BWDSTART = FALSE
LDAT_ACT = LCPDAT38
FDAT_ACT = FP129
BAS(#CP_PARAMS, ATBg_BAS_VELDefinition)
LIN XP129
Arc_Off(1, AC_WDAT71)
;ENDFOLD
;FOLD PTP P130 CONT Vel=100 % PDAT95 Tool[1]:TOCH Base[0];%{PE}%R 8.3.48,%MKUKATPBASIS,%CMOVE,%VPTP,%P 1:PTP, 2:P130, 3:C_DIS, 5:100, 7:PDAT95
$BWDSTART=FALSE
PDAT_ACT=PPDAT95
FDAT_ACT=FP130
BAS(#PTP_PARAMS,100)
PTP XP130 C_DIS
;ENDFOLD
;FOLD PTP P131 CONT Vel=100 % PDAT96 Tool[1]:TOCH Base[0];%{PE}%R 8.3.48,%MKUKATPBASIS,%CMOVE,%VPTP,%P 1:PTP, 2:P131, 3:C_DIS, 5:100, 7:PDAT96
$BWDSTART=FALSE
PDAT_ACT=PPDAT96
FDAT_ACT=FP131
BAS(#PTP_PARAMS,100)
PTP XP131 C_DIS
;ENDFOLD
;FOLD ; CORDAO 17;%{PE}%R 8.3.48,%MKUKATPBASIS,%CCOMMENT,%VNORMAL,%P 2:CORDAO 17
;ENDFOLD
;FOLD ARCON WDAT72 PTP P132 Vel=100 % PDAT97 Tool[1]:TOCH Base[0] ;%{PE}
;FOLD Parameters ;%{h}
;Params IlfProvider=kukaroboter.arctech.arconptp; Kuka.PointName=P132; Kuka.BlendingEnabled=False; Kuka.MoveDataPtpName=PDAT97; Kuka.VelocityPtp=100; Kuka.MovementParameterFieldEnabled=True; ArcTech.WdatVarName=WDAT72; ArcTech.SeamName=
;ENDFOLD
$BWDSTART = FALSE
PDAT_ACT = PPDAT97
FDAT_ACT = FP132
BAS(#PTP_PARAMS, 100.0)
TRIGGER WHEN DISTANCE = 1 DELAY = ATBg_PreDefinitionTime DO Arc_DefineStrikeParams(1, AS_WDAT72) PRIO = -1
Arc_DefineCpPattern(#OffInAdvance, WV_WDAT72, TRUE)
PTP XP132
Arc_On(1, AS_WDAT72, ATBg_StartErrSetField[1], AW_WDAT72, WV_WDAT72, ATBg_WeldErrSetField[1], #StdArcOn, " ")
Arc_DefineCpPattern(#OnInAdvance, WV_WDAT72, TRUE)
;ENDFOLD
;FOLD ARCOFF WDAT73 LIN P133 CPDAT39 Tool[1]:TOCH Base[0] ;%{PE}
;FOLD Parameters ;%{h}
;Params IlfProvider=kukaroboter.arctech.arcofflin; Kuka.PointName=P133; Kuka.BlendingEnabled=False; Kuka.MoveDataName=CPDAT39;  Kuka.MovementParameterFieldEnabled=True; ArcTech.WdatVarName=WDAT73
;ENDFOLD
$BWDSTART = FALSE
LDAT_ACT = LCPDAT39
FDAT_ACT = FP133
BAS(#CP_PARAMS, ATBg_BAS_VELDefinition)
LIN XP133
Arc_Off(1, AC_WDAT73)
;ENDFOLD
;FOLD PTP P143 CONT Vel=100 % PDAT106 Tool[1]:TOCH Base[0];%{PE}%R 8.3.48,%MKUKATPBASIS,%CMOVE,%VPTP,%P 1:PTP, 2:P143, 3:C_DIS, 5:100, 7:PDAT106
$BWDSTART=FALSE
PDAT_ACT=PPDAT106
FDAT_ACT=FP143
BAS(#PTP_PARAMS,100)
PTP XP143 C_DIS
;ENDFOLD
;FOLD PTP P144 CONT Vel=100 % PDAT107 Tool[1]:TOCH Base[0];%{PE}%R 8.3.48,%MKUKATPBASIS,%CMOVE,%VPTP,%P 1:PTP, 2:P144, 3:C_DIS, 5:100, 7:PDAT107
$BWDSTART=FALSE
PDAT_ACT=PPDAT107
FDAT_ACT=FP144
BAS(#PTP_PARAMS,100)
PTP XP144 C_DIS
;ENDFOLD
;FOLD ; CORDAO 18;%{PE}%R 8.3.48,%MKUKATPBASIS,%CCOMMENT,%VNORMAL,%P 2:CORDAO 18
;ENDFOLD
;FOLD ARCON WDAT74 PTP P134 Vel=100 % PDAT98 Tool[1]:TOCH Base[0] ;%{PE}
;FOLD Parameters ;%{h}
;Params IlfProvider=kukaroboter.arctech.arconptp; Kuka.PointName=P134; Kuka.BlendingEnabled=False; Kuka.MoveDataPtpName=PDAT98; Kuka.VelocityPtp=100; Kuka.MovementParameterFieldEnabled=True; ArcTech.WdatVarName=WDAT74; ArcTech.SeamName=
;ENDFOLD
$BWDSTART = FALSE
PDAT_ACT = PPDAT98
FDAT_ACT = FP134
BAS(#PTP_PARAMS, 100.0)
TRIGGER WHEN DISTANCE = 1 DELAY = ATBg_PreDefinitionTime DO Arc_DefineStrikeParams(1, AS_WDAT74) PRIO = -1
Arc_DefineCpPattern(#OffInAdvance, WV_WDAT74, TRUE)
PTP XP134
Arc_On(1, AS_WDAT74, ATBg_StartErrSetField[1], AW_WDAT74, WV_WDAT74, ATBg_WeldErrSetField[1], #StdArcOn, " ")
Arc_DefineCpPattern(#OnInAdvance, WV_WDAT74, TRUE)
;ENDFOLD
;FOLD ARCOFF WDAT75 LIN P135 CPDAT40 Tool[1]:TOCH Base[0] ;%{PE}
;FOLD Parameters ;%{h}
;Params IlfProvider=kukaroboter.arctech.arcofflin; Kuka.PointName=P135; Kuka.BlendingEnabled=False; Kuka.MoveDataName=CPDAT40;  Kuka.MovementParameterFieldEnabled=True; ArcTech.WdatVarName=WDAT75
;ENDFOLD
$BWDSTART = FALSE
LDAT_ACT = LCPDAT40
FDAT_ACT = FP135
BAS(#CP_PARAMS, ATBg_BAS_VELDefinition)
LIN XP135
Arc_Off(1, AC_WDAT75)
;ENDFOLD
;FOLD PTP P137 CONT Vel=100 % PDAT100 Tool[1]:TOCH Base[0];%{PE}%R 8.3.48,%MKUKATPBASIS,%CMOVE,%VPTP,%P 1:PTP, 2:P137, 3:C_DIS, 5:100, 7:PDAT100
$BWDSTART=FALSE
PDAT_ACT=PPDAT100
FDAT_ACT=FP137
BAS(#PTP_PARAMS,100)
PTP XP137 C_DIS
;ENDFOLD
;FOLD PTP P136 CONT Vel=100 % PDAT99 Tool[1]:TOCH Base[0];%{PE}%R 8.3.48,%MKUKATPBASIS,%CMOVE,%VPTP,%P 1:PTP, 2:P136, 3:C_DIS, 5:100, 7:PDAT99
$BWDSTART=FALSE
PDAT_ACT=PPDAT99
FDAT_ACT=FP136
BAS(#PTP_PARAMS,100)
PTP XP136 C_DIS
;ENDFOLD
;FOLD ; CORDAO 19;%{PE}%R 8.3.48,%MKUKATPBASIS,%CCOMMENT,%VNORMAL,%P 2:CORDAO 19
;ENDFOLD
;FOLD ARCON WDAT76 PTP P145 Vel=100 % PDAT108 Tool[1]:TOCH Base[0] ;%{PE}
;FOLD Parameters ;%{h}
;Params IlfProvider=kukaroboter.arctech.arconptp; Kuka.PointName=P145; Kuka.BlendingEnabled=False; Kuka.MoveDataPtpName=PDAT108; Kuka.VelocityPtp=100; Kuka.MovementParameterFieldEnabled=True; ArcTech.WdatVarName=WDAT76; ArcTech.SeamName=
;ENDFOLD
$BWDSTART = FALSE
PDAT_ACT = PPDAT108
FDAT_ACT = FP145
BAS(#PTP_PARAMS, 100.0)
TRIGGER WHEN DISTANCE = 1 DELAY = ATBg_PreDefinitionTime DO Arc_DefineStrikeParams(1, AS_WDAT76) PRIO = -1
Arc_DefineCpPattern(#OffInAdvance, WV_WDAT76, TRUE)
PTP XP145
Arc_On(1, AS_WDAT76, ATBg_StartErrSetField[1], AW_WDAT76, WV_WDAT76, ATBg_WeldErrSetField[1], #StdArcOn, " ")
Arc_DefineCpPattern(#OnInAdvance, WV_WDAT76, TRUE)
;ENDFOLD
;FOLD ARCOFF WDAT77 LIN P146 CPDAT41 Tool[1]:TOCH Base[0] ;%{PE}
;FOLD Parameters ;%{h}
;Params IlfProvider=kukaroboter.arctech.arcofflin; Kuka.PointName=P146; Kuka.BlendingEnabled=False; Kuka.MoveDataName=CPDAT41;  Kuka.MovementParameterFieldEnabled=True; ArcTech.WdatVarName=WDAT77
;ENDFOLD
$BWDSTART = FALSE
LDAT_ACT = LCPDAT41
FDAT_ACT = FP146
BAS(#CP_PARAMS, ATBg_BAS_VELDefinition)
LIN XP146
Arc_Off(1, AC_WDAT77)
;ENDFOLD
;FOLD PTP P157 CONT Vel=100 % PDAT115 Tool[1]:TOCH Base[0];%{PE}%R 8.3.48,%MKUKATPBASIS,%CMOVE,%VPTP,%P 1:PTP, 2:P157, 3:C_DIS, 5:100, 7:PDAT115
$BWDSTART=FALSE
PDAT_ACT=PPDAT115
FDAT_ACT=FP157
BAS(#PTP_PARAMS,100)
PTP XP157 C_DIS
;ENDFOLD
;FOLD PTP P158 CONT Vel=100 % PDAT116 Tool[1]:TOCH Base[0];%{PE}%R 8.3.48,%MKUKATPBASIS,%CMOVE,%VPTP,%P 1:PTP, 2:P158, 3:C_DIS, 5:100, 7:PDAT116
$BWDSTART=FALSE
PDAT_ACT=PPDAT116
FDAT_ACT=FP158
BAS(#PTP_PARAMS,100)
PTP XP158 C_DIS
;ENDFOLD
;FOLD PTP P159 CONT Vel=100 % PDAT117 Tool[1]:TOCH Base[0];%{PE}%R 8.3.48,%MKUKATPBASIS,%CMOVE,%VPTP,%P 1:PTP, 2:P159, 3:C_DIS, 5:100, 7:PDAT117
$BWDSTART=FALSE
PDAT_ACT=PPDAT117
FDAT_ACT=FP159
BAS(#PTP_PARAMS,100)
PTP XP159 C_DIS
;ENDFOLD
;FOLD ; CORDAO 20;%{PE}%R 8.3.48,%MKUKATPBASIS,%CCOMMENT,%VNORMAL,%P 2:CORDAO 20
;ENDFOLD
;FOLD ARCON WDAT78 PTP P147 Vel=100 % PDAT109 Tool[1]:TOCH Base[0] ;%{PE}
;FOLD Parameters ;%{h}
;Params IlfProvider=kukaroboter.arctech.arconptp; Kuka.PointName=P147; Kuka.BlendingEnabled=False; Kuka.MoveDataPtpName=PDAT109; Kuka.VelocityPtp=100; Kuka.MovementParameterFieldEnabled=True; ArcTech.WdatVarName=WDAT78; ArcTech.SeamName=
;ENDFOLD
$BWDSTART = FALSE
PDAT_ACT = PPDAT109
FDAT_ACT = FP147
BAS(#PTP_PARAMS, 100.0)
TRIGGER WHEN DISTANCE = 1 DELAY = ATBg_PreDefinitionTime DO Arc_DefineStrikeParams(1, AS_WDAT78) PRIO = -1
Arc_DefineCpPattern(#OffInAdvance, WV_WDAT78, TRUE)
PTP XP147
Arc_On(1, AS_WDAT78, ATBg_StartErrSetField[1], AW_WDAT78, WV_WDAT78, ATBg_WeldErrSetField[1], #StdArcOn, " ")
Arc_DefineCpPattern(#OnInAdvance, WV_WDAT78, TRUE)
;ENDFOLD
;FOLD ARCOFF WDAT87 LIN P160 CPDAT46 Tool[1]:TOCH Base[0] ;%{PE}
;FOLD Parameters ;%{h}
;Params IlfProvider=kukaroboter.arctech.arcofflin; Kuka.PointName=P160; Kuka.BlendingEnabled=False; Kuka.MoveDataName=CPDAT46;  Kuka.MovementParameterFieldEnabled=True; ArcTech.WdatVarName=WDAT87
;ENDFOLD
$BWDSTART = FALSE
LDAT_ACT = LCPDAT46
FDAT_ACT = FP160
BAS(#CP_PARAMS, ATBg_BAS_VELDefinition)
LIN XP160
Arc_Off(1, AC_WDAT87)
;ENDFOLD
;FOLD PTP P161 CONT Vel=100 % PDAT118 Tool[1]:TOCH Base[0];%{PE}%R 8.3.48,%MKUKATPBASIS,%CMOVE,%VPTP,%P 1:PTP, 2:P161, 3:C_DIS, 5:100, 7:PDAT118
$BWDSTART=FALSE
PDAT_ACT=PPDAT118
FDAT_ACT=FP161
BAS(#PTP_PARAMS,100)
PTP XP161 C_DIS
;ENDFOLD
;FOLD PTP P162 CONT Vel=100 % PDAT119 Tool[1]:TOCH Base[0];%{PE}%R 8.3.48,%MKUKATPBASIS,%CMOVE,%VPTP,%P 1:PTP, 2:P162, 3:C_DIS, 5:100, 7:PDAT119
$BWDSTART=FALSE
PDAT_ACT=PPDAT119
FDAT_ACT=FP162
BAS(#PTP_PARAMS,100)
PTP XP162 C_DIS
;ENDFOLD
;FOLD ; CORDAO 20;%{PE}%R 8.3.48,%MKUKATPBASIS,%CCOMMENT,%VNORMAL,%P 2:CORDAO 20
;ENDFOLD
;FOLD ARCON WDAT79 PTP P148 Vel=100 % PDAT110 Tool[1]:TOCH Base[0] ;%{PE}
;FOLD Parameters ;%{h}
;Params IlfProvider=kukaroboter.arctech.arconptp; Kuka.PointName=P148; Kuka.BlendingEnabled=False; Kuka.MoveDataPtpName=PDAT110; Kuka.VelocityPtp=100; Kuka.MovementParameterFieldEnabled=True; ArcTech.WdatVarName=WDAT79; ArcTech.SeamName=
;ENDFOLD
$BWDSTART = FALSE
PDAT_ACT = PPDAT110
FDAT_ACT = FP148
BAS(#PTP_PARAMS, 100.0)
TRIGGER WHEN DISTANCE = 1 DELAY = ATBg_PreDefinitionTime DO Arc_DefineStrikeParams(1, AS_WDAT79) PRIO = -1
Arc_DefineCpPattern(#OffInAdvance, WV_WDAT79, TRUE)
PTP XP148
Arc_On(1, AS_WDAT79, ATBg_StartErrSetField[1], AW_WDAT79, WV_WDAT79, ATBg_WeldErrSetField[1], #StdArcOn, " ")
Arc_DefineCpPattern(#OnInAdvance, WV_WDAT79, TRUE)
;ENDFOLD
;FOLD ARCOFF WDAT80 LIN P149 CPDAT42 Tool[1]:TOCH Base[0] ;%{PE}
;FOLD Parameters ;%{h}
;Params IlfProvider=kukaroboter.arctech.arcofflin; Kuka.PointName=P149; Kuka.BlendingEnabled=False; Kuka.MoveDataName=CPDAT42;  Kuka.MovementParameterFieldEnabled=True; ArcTech.WdatVarName=WDAT80
;ENDFOLD
$BWDSTART = FALSE
LDAT_ACT = LCPDAT42
FDAT_ACT = FP149
BAS(#CP_PARAMS, ATBg_BAS_VELDefinition)
LIN XP149
Arc_Off(1, AC_WDAT80)
;ENDFOLD
;FOLD PTP P163 CONT Vel=100 % PDAT120 Tool[1]:TOCH Base[0];%{PE}%R 8.3.48,%MKUKATPBASIS,%CMOVE,%VPTP,%P 1:PTP, 2:P163, 3:C_DIS, 5:100, 7:PDAT120
$BWDSTART=FALSE
PDAT_ACT=PPDAT120
FDAT_ACT=FP163
BAS(#PTP_PARAMS,100)
PTP XP163 C_DIS
;ENDFOLD
;FOLD PTP P164 CONT Vel=100 % PDAT121 Tool[1]:TOCH Base[0];%{PE}%R 8.3.48,%MKUKATPBASIS,%CMOVE,%VPTP,%P 1:PTP, 2:P164, 3:C_DIS, 5:100, 7:PDAT121
$BWDSTART=FALSE
PDAT_ACT=PPDAT121
FDAT_ACT=FP164
BAS(#PTP_PARAMS,100)
PTP XP164 C_DIS
;ENDFOLD
;FOLD ; CORDAO 21;%{PE}%R 8.3.48,%MKUKATPBASIS,%CCOMMENT,%VNORMAL,%P 2:CORDAO 21
;ENDFOLD
;FOLD ARCON WDAT83 PTP P152 Vel=100 % PDAT112 Tool[1]:TOCH Base[0] ;%{PE}
;FOLD Parameters ;%{h}
;Params IlfProvider=kukaroboter.arctech.arconptp; Kuka.PointName=P152; Kuka.BlendingEnabled=False; Kuka.MoveDataPtpName=PDAT112; Kuka.VelocityPtp=100; Kuka.MovementParameterFieldEnabled=True; ArcTech.WdatVarName=WDAT83; ArcTech.SeamName=
;ENDFOLD
$BWDSTART = FALSE
PDAT_ACT = PPDAT112
FDAT_ACT = FP152
BAS(#PTP_PARAMS, 100.0)
TRIGGER WHEN DISTANCE = 1 DELAY = ATBg_PreDefinitionTime DO Arc_DefineStrikeParams(1, AS_WDAT83) PRIO = -1
Arc_DefineCpPattern(#OffInAdvance, WV_WDAT83, TRUE)
PTP XP152
Arc_On(1, AS_WDAT83, ATBg_StartErrSetField[1], AW_WDAT83, WV_WDAT83, ATBg_WeldErrSetField[1], #StdArcOn, " ")
Arc_DefineCpPattern(#OnInAdvance, WV_WDAT83, TRUE)
;ENDFOLD
;FOLD ARCOFF WDAT84 LIN P153 CPDAT44 Tool[1]:TOCH Base[0] ;%{PE}
;FOLD Parameters ;%{h}
;Params IlfProvider=kukaroboter.arctech.arcofflin; Kuka.PointName=P153; Kuka.BlendingEnabled=False; Kuka.MoveDataName=CPDAT44;  Kuka.MovementParameterFieldEnabled=True; ArcTech.WdatVarName=WDAT84
;ENDFOLD
$BWDSTART = FALSE
LDAT_ACT = LCPDAT44
FDAT_ACT = FP153
BAS(#CP_PARAMS, ATBg_BAS_VELDefinition)
LIN XP153
Arc_Off(1, AC_WDAT84)
;ENDFOLD
;FOLD PTP P165 CONT Vel=100 % PDAT122 Tool[1]:TOCH Base[0];%{PE}%R 8.3.48,%MKUKATPBASIS,%CMOVE,%VPTP,%P 1:PTP, 2:P165, 3:C_DIS, 5:100, 7:PDAT122
$BWDSTART=FALSE
PDAT_ACT=PPDAT122
FDAT_ACT=FP165
BAS(#PTP_PARAMS,100)
PTP XP165 C_DIS
;ENDFOLD
;FOLD PTP P166 CONT Vel=100 % PDAT123 Tool[1]:TOCH Base[0];%{PE}%R 8.3.48,%MKUKATPBASIS,%CMOVE,%VPTP,%P 1:PTP, 2:P166, 3:C_DIS, 5:100, 7:PDAT123
$BWDSTART=FALSE
PDAT_ACT=PPDAT123
FDAT_ACT=FP166
BAS(#PTP_PARAMS,100)
PTP XP166 C_DIS
;ENDFOLD
;FOLD ; CORDAO 22;%{PE}%R 8.3.48,%MKUKATPBASIS,%CCOMMENT,%VNORMAL,%P 2:CORDAO 22
;ENDFOLD
;FOLD ARCON WDAT85 PTP P154 Vel=100 % PDAT113 Tool[1]:TOCH Base[0] ;%{PE}
;FOLD Parameters ;%{h}
;Params IlfProvider=kukaroboter.arctech.arconptp; Kuka.PointName=P154; Kuka.BlendingEnabled=False; Kuka.MoveDataPtpName=PDAT113; Kuka.VelocityPtp=100; Kuka.MovementParameterFieldEnabled=True; ArcTech.WdatVarName=WDAT85; ArcTech.SeamName=
;ENDFOLD
$BWDSTART = FALSE
PDAT_ACT = PPDAT113
FDAT_ACT = FP154
BAS(#PTP_PARAMS, 100.0)
TRIGGER WHEN DISTANCE = 1 DELAY = ATBg_PreDefinitionTime DO Arc_DefineStrikeParams(1, AS_WDAT85) PRIO = -1
Arc_DefineCpPattern(#OffInAdvance, WV_WDAT85, TRUE)
PTP XP154
Arc_On(1, AS_WDAT85, ATBg_StartErrSetField[1], AW_WDAT85, WV_WDAT85, ATBg_WeldErrSetField[1], #StdArcOn, " ")
Arc_DefineCpPattern(#OnInAdvance, WV_WDAT85, TRUE)
;ENDFOLD
;FOLD ARCOFF WDAT86 LIN P155 CPDAT45 Tool[1]:TOCH Base[0] ;%{PE}
;FOLD Parameters ;%{h}
;Params IlfProvider=kukaroboter.arctech.arcofflin; Kuka.PointName=P155; Kuka.BlendingEnabled=False; Kuka.MoveDataName=CPDAT45;  Kuka.MovementParameterFieldEnabled=True; ArcTech.WdatVarName=WDAT86
;ENDFOLD
$BWDSTART = FALSE
LDAT_ACT = LCPDAT45
FDAT_ACT = FP155
BAS(#CP_PARAMS, ATBg_BAS_VELDefinition)
LIN XP155
Arc_Off(1, AC_WDAT86)
;ENDFOLD
;FOLD PTP P156 CONT Vel=100 % PDAT114 Tool[1]:TOCH Base[0];%{PE}%R 8.3.48,%MKUKATPBASIS,%CMOVE,%VPTP,%P 1:PTP, 2:P156, 3:C_DIS, 5:100, 7:PDAT114
$BWDSTART=FALSE
PDAT_ACT=PPDAT114
FDAT_ACT=FP156
BAS(#PTP_PARAMS,100)
PTP XP156 C_DIS
;ENDFOLD
;FOLD PTP P169 CONT Vel=100 % PDAT125 Tool[1]:TOCH Base[0];%{PE}%R 8.3.48,%MKUKATPBASIS,%CMOVE,%VPTP,%P 1:PTP, 2:P169, 3:C_DIS, 5:100, 7:PDAT125
$BWDSTART=FALSE
PDAT_ACT=PPDAT125
FDAT_ACT=FP169
BAS(#PTP_PARAMS,100)
PTP XP169 C_DIS
;ENDFOLD
;FOLD ; CORDAO 21;%{PE}%R 8.3.48,%MKUKATPBASIS,%CCOMMENT,%VNORMAL,%P 2:CORDAO 21
;ENDFOLD
;FOLD ARCON WDAT88 PTP P167 Vel=100 % PDAT124 Tool[1]:TOCH Base[0] ;%{PE}
;FOLD Parameters ;%{h}
;Params IlfProvider=kukaroboter.arctech.arconptp; Kuka.PointName=P167; Kuka.BlendingEnabled=False; Kuka.MoveDataPtpName=PDAT124; Kuka.VelocityPtp=100; Kuka.MovementParameterFieldEnabled=True; ArcTech.WdatVarName=WDAT88; ArcTech.SeamName=
;ENDFOLD
$BWDSTART = FALSE
PDAT_ACT = PPDAT124
FDAT_ACT = FP167
BAS(#PTP_PARAMS, 100.0)
TRIGGER WHEN DISTANCE = 1 DELAY = ATBg_PreDefinitionTime DO Arc_DefineStrikeParams(1, AS_WDAT88) PRIO = -1
Arc_DefineCpPattern(#OffInAdvance, WV_WDAT88, TRUE)
PTP XP167
Arc_On(1, AS_WDAT88, ATBg_StartErrSetField[1], AW_WDAT88, WV_WDAT88, ATBg_WeldErrSetField[1], #StdArcOn, " ")
Arc_DefineCpPattern(#OnInAdvance, WV_WDAT88, TRUE)
;ENDFOLD
;FOLD ARCOFF WDAT89 LIN P168 CPDAT47 Tool[1]:TOCH Base[0] ;%{PE}
;FOLD Parameters ;%{h}
;Params IlfProvider=kukaroboter.arctech.arcofflin; Kuka.PointName=P168; Kuka.BlendingEnabled=False; Kuka.MoveDataName=CPDAT47;  Kuka.MovementParameterFieldEnabled=True; ArcTech.WdatVarName=WDAT89
;ENDFOLD
$BWDSTART = FALSE
LDAT_ACT = LCPDAT47
FDAT_ACT = FP168
BAS(#CP_PARAMS, ATBg_BAS_VELDefinition)
LIN XP168
Arc_Off(1, AC_WDAT89)
;ENDFOLD
;FOLD PTP P173 CONT Vel=100 % PDAT128 Tool[1]:TOCH Base[0];%{PE}%R 8.3.48,%MKUKATPBASIS,%CMOVE,%VPTP,%P 1:PTP, 2:P173, 3:C_DIS, 5:100, 7:PDAT128
$BWDSTART=FALSE
PDAT_ACT=PPDAT128
FDAT_ACT=FP173
BAS(#PTP_PARAMS,100)
PTP XP173 C_DIS
;ENDFOLD
;FOLD PTP P172 CONT Vel=100 % PDAT127 Tool[1]:TOCH Base[0];%{PE}%R 8.3.48,%MKUKATPBASIS,%CMOVE,%VPTP,%P 1:PTP, 2:P172, 3:C_DIS, 5:100, 7:PDAT127
$BWDSTART=FALSE
PDAT_ACT=PPDAT127
FDAT_ACT=FP172
BAS(#PTP_PARAMS,100)
PTP XP172 C_DIS
;ENDFOLD
;FOLD ; CORDAO 21;%{PE}%R 8.3.48,%MKUKATPBASIS,%CCOMMENT,%VNORMAL,%P 2:CORDAO 21
;ENDFOLD
;FOLD ARCON WDAT90 PTP P170 Vel=100 % PDAT126 Tool[1]:TOCH Base[0] ;%{PE}
;FOLD Parameters ;%{h}
;Params IlfProvider=kukaroboter.arctech.arconptp; Kuka.PointName=P170; Kuka.BlendingEnabled=False; Kuka.MoveDataPtpName=PDAT126; Kuka.VelocityPtp=100; Kuka.MovementParameterFieldEnabled=True; ArcTech.WdatVarName=WDAT90; ArcTech.SeamName=
;ENDFOLD
$BWDSTART = FALSE
PDAT_ACT = PPDAT126
FDAT_ACT = FP170
BAS(#PTP_PARAMS, 100.0)
TRIGGER WHEN DISTANCE = 1 DELAY = ATBg_PreDefinitionTime DO Arc_DefineStrikeParams(1, AS_WDAT90) PRIO = -1
Arc_DefineCpPattern(#OffInAdvance, WV_WDAT90, TRUE)
PTP XP170
Arc_On(1, AS_WDAT90, ATBg_StartErrSetField[1], AW_WDAT90, WV_WDAT90, ATBg_WeldErrSetField[1], #StdArcOn, " ")
Arc_DefineCpPattern(#OnInAdvance, WV_WDAT90, TRUE)
;ENDFOLD
;FOLD ARCOFF WDAT91 LIN P171 CPDAT48 Tool[1]:TOCH Base[0] ;%{PE}
;FOLD Parameters ;%{h}
;Params IlfProvider=kukaroboter.arctech.arcofflin; Kuka.PointName=P171; Kuka.BlendingEnabled=False; Kuka.MoveDataName=CPDAT48;  Kuka.MovementParameterFieldEnabled=True; ArcTech.WdatVarName=WDAT91
;ENDFOLD
$BWDSTART = FALSE
LDAT_ACT = LCPDAT48
FDAT_ACT = FP171
BAS(#CP_PARAMS, ATBg_BAS_VELDefinition)
LIN XP171
Arc_Off(1, AC_WDAT91)
;ENDFOLD
;FOLD PTP P174 CONT Vel=100 % PDAT129 Tool[1]:TOCH Base[0];%{PE}%R 8.3.48,%MKUKATPBASIS,%CMOVE,%VPTP,%P 1:PTP, 2:P174, 3:C_DIS, 5:100, 7:PDAT129
$BWDSTART=FALSE
PDAT_ACT=PPDAT129
FDAT_ACT=FP174
BAS(#PTP_PARAMS,100)
PTP XP174 C_DIS
;ENDFOLD
;FOLD PTP P185 CONT Vel=100 % PDAT137 Tool[1]:TOCH Base[0];%{PE}%R 8.3.48,%MKUKATPBASIS,%CMOVE,%VPTP,%P 1:PTP, 2:P185, 3:C_DIS, 5:100, 7:PDAT137
$BWDSTART=FALSE
PDAT_ACT=PPDAT137
FDAT_ACT=FP185
BAS(#PTP_PARAMS,100)
PTP XP185 C_DIS
;ENDFOLD
;FOLD ; CORDAO 21;%{PE}%R 8.3.48,%MKUKATPBASIS,%CCOMMENT,%VNORMAL,%P 2:CORDAO 21
;ENDFOLD
;FOLD ARCON WDAT92 PTP P175 Vel=100 % PDAT130 Tool[1]:TOCH Base[0] ;%{PE}
;FOLD Parameters ;%{h}
;Params IlfProvider=kukaroboter.arctech.arconptp; Kuka.PointName=P175; Kuka.BlendingEnabled=False; Kuka.MoveDataPtpName=PDAT130; Kuka.VelocityPtp=100; Kuka.MovementParameterFieldEnabled=True; ArcTech.WdatVarName=WDAT92; ArcTech.SeamName=
;ENDFOLD
$BWDSTART = FALSE
PDAT_ACT = PPDAT130
FDAT_ACT = FP175
BAS(#PTP_PARAMS, 100.0)
TRIGGER WHEN DISTANCE = 1 DELAY = ATBg_PreDefinitionTime DO Arc_DefineStrikeParams(1, AS_WDAT92) PRIO = -1
Arc_DefineCpPattern(#OffInAdvance, WV_WDAT92, TRUE)
PTP XP175
Arc_On(1, AS_WDAT92, ATBg_StartErrSetField[1], AW_WDAT92, WV_WDAT92, ATBg_WeldErrSetField[1], #StdArcOn, " ")
Arc_DefineCpPattern(#OnInAdvance, WV_WDAT92, TRUE)
;ENDFOLD
;FOLD ARCOFF WDAT93 LIN P176 CPDAT49 Tool[1]:TOCH Base[0] ;%{PE}
;FOLD Parameters ;%{h}
;Params IlfProvider=kukaroboter.arctech.arcofflin; Kuka.PointName=P176; Kuka.BlendingEnabled=False; Kuka.MoveDataName=CPDAT49;  Kuka.MovementParameterFieldEnabled=True; ArcTech.WdatVarName=WDAT93
;ENDFOLD
$BWDSTART = FALSE
LDAT_ACT = LCPDAT49
FDAT_ACT = FP176
BAS(#CP_PARAMS, ATBg_BAS_VELDefinition)
LIN XP176
Arc_Off(1, AC_WDAT93)
;ENDFOLD
;FOLD PTP P184 CONT Vel=100 % PDAT136 Tool[1]:TOCH Base[0];%{PE}%R 8.3.48,%MKUKATPBASIS,%CMOVE,%VPTP,%P 1:PTP, 2:P184, 3:C_DIS, 5:100, 7:PDAT136
$BWDSTART=FALSE
PDAT_ACT=PPDAT136
FDAT_ACT=FP184
BAS(#PTP_PARAMS,100)
PTP XP184 C_DIS
;ENDFOLD
;FOLD ; CORDAO 21;%{PE}%R 8.3.48,%MKUKATPBASIS,%CCOMMENT,%VNORMAL,%P 2:CORDAO 21
;ENDFOLD
;FOLD ARCON WDAT94 PTP P177 Vel=100 % PDAT131 Tool[1]:TOCH Base[0] ;%{PE}
;FOLD Parameters ;%{h}
;Params IlfProvider=kukaroboter.arctech.arconptp; Kuka.PointName=P177; Kuka.BlendingEnabled=False; Kuka.MoveDataPtpName=PDAT131; Kuka.VelocityPtp=100; Kuka.MovementParameterFieldEnabled=True; ArcTech.WdatVarName=WDAT94; ArcTech.SeamName=
;ENDFOLD
$BWDSTART = FALSE
PDAT_ACT = PPDAT131
FDAT_ACT = FP177
BAS(#PTP_PARAMS, 100.0)
TRIGGER WHEN DISTANCE = 1 DELAY = ATBg_PreDefinitionTime DO Arc_DefineStrikeParams(1, AS_WDAT94) PRIO = -1
Arc_DefineCpPattern(#OffInAdvance, WV_WDAT94, TRUE)
PTP XP177
Arc_On(1, AS_WDAT94, ATBg_StartErrSetField[1], AW_WDAT94, WV_WDAT94, ATBg_WeldErrSetField[1], #StdArcOn, " ")
Arc_DefineCpPattern(#OnInAdvance, WV_WDAT94, TRUE)
;ENDFOLD
;FOLD ARCOFF WDAT95 LIN P178 CPDAT50 Tool[1]:TOCH Base[0] ;%{PE}
;FOLD Parameters ;%{h}
;Params IlfProvider=kukaroboter.arctech.arcofflin; Kuka.PointName=P178; Kuka.BlendingEnabled=False; Kuka.MoveDataName=CPDAT50;  Kuka.MovementParameterFieldEnabled=True; ArcTech.WdatVarName=WDAT95
;ENDFOLD
$BWDSTART = FALSE
LDAT_ACT = LCPDAT50
FDAT_ACT = FP178
BAS(#CP_PARAMS, ATBg_BAS_VELDefinition)
LIN XP178
Arc_Off(1, AC_WDAT95)
;ENDFOLD
;FOLD PTP P179 CONT Vel=100 % PDAT132 Tool[1]:TOCH Base[0];%{PE}%R 8.3.48,%MKUKATPBASIS,%CMOVE,%VPTP,%P 1:PTP, 2:P179, 3:C_DIS, 5:100, 7:PDAT132
$BWDSTART=FALSE
PDAT_ACT=PPDAT132
FDAT_ACT=FP179
BAS(#PTP_PARAMS,100)
PTP XP179 C_DIS
;ENDFOLD
;FOLD PTP P183 CONT Vel=100 % PDAT135 Tool[1]:TOCH Base[0];%{PE}%R 8.3.48,%MKUKATPBASIS,%CMOVE,%VPTP,%P 1:PTP, 2:P183, 3:C_DIS, 5:100, 7:PDAT135
$BWDSTART=FALSE
PDAT_ACT=PPDAT135
FDAT_ACT=FP183
BAS(#PTP_PARAMS,100)
PTP XP183 C_DIS
;ENDFOLD
;FOLD ; CORDAO 21;%{PE}%R 8.3.48,%MKUKATPBASIS,%CCOMMENT,%VNORMAL,%P 2:CORDAO 21
;ENDFOLD
;FOLD ARCON WDAT96 PTP P180 Vel=100 % PDAT133 Tool[1]:TOCH Base[0] ;%{PE}
;FOLD Parameters ;%{h}
;Params IlfProvider=kukaroboter.arctech.arconptp; Kuka.PointName=P180; Kuka.BlendingEnabled=False; Kuka.MoveDataPtpName=PDAT133; Kuka.VelocityPtp=100; Kuka.MovementParameterFieldEnabled=True; ArcTech.WdatVarName=WDAT96; ArcTech.SeamName=
;ENDFOLD
$BWDSTART = FALSE
PDAT_ACT = PPDAT133
FDAT_ACT = FP180
BAS(#PTP_PARAMS, 100.0)
TRIGGER WHEN DISTANCE = 1 DELAY = ATBg_PreDefinitionTime DO Arc_DefineStrikeParams(1, AS_WDAT96) PRIO = -1
Arc_DefineCpPattern(#OffInAdvance, WV_WDAT96, TRUE)
PTP XP180
Arc_On(1, AS_WDAT96, ATBg_StartErrSetField[1], AW_WDAT96, WV_WDAT96, ATBg_WeldErrSetField[1], #StdArcOn, " ")
Arc_DefineCpPattern(#OnInAdvance, WV_WDAT96, TRUE)
;ENDFOLD
;FOLD ARCOFF WDAT97 LIN P181 CPDAT51 Tool[1]:TOCH Base[0] ;%{PE}
;FOLD Parameters ;%{h}
;Params IlfProvider=kukaroboter.arctech.arcofflin; Kuka.PointName=P181; Kuka.BlendingEnabled=False; Kuka.MoveDataName=CPDAT51;  Kuka.MovementParameterFieldEnabled=True; ArcTech.WdatVarName=WDAT97
;ENDFOLD
$BWDSTART = FALSE
LDAT_ACT = LCPDAT51
FDAT_ACT = FP181
BAS(#CP_PARAMS, ATBg_BAS_VELDefinition)
LIN XP181
Arc_Off(1, AC_WDAT97)
;ENDFOLD
;FOLD PTP P182 CONT Vel=100 % PDAT134 Tool[1]:TOCH Base[0];%{PE}%R 8.3.48,%MKUKATPBASIS,%CMOVE,%VPTP,%P 1:PTP, 2:P182, 3:C_DIS, 5:100, 7:PDAT134
$BWDSTART=FALSE
PDAT_ACT=PPDAT134
FDAT_ACT=FP182
BAS(#PTP_PARAMS,100)
PTP XP182 C_DIS
;ENDFOLD
;FOLD PTP HOME Vel=100 % DEFAULT;%{PE}%R 8.3.48,%MKUKATPBASIS,%CMOVE,%VPTP,%P 1:PTP, 2:HOME, 3:, 5:100, 7:DEFAULT
$BWDSTART=FALSE
PDAT_ACT=PDEFAULT
FDAT_ACT=FHOME
BAS(#PTP_PARAMS,100)
$H_POS=XHOME
PTP XHOME
;ENDFOLD
;FOLD WAIT FOR NOT ( IN 129 'AVA/REC MESA B' );%{PE}%R 8.3.48,%MKUKATPBASIS,%CEXT_WAIT_FOR,%VEXT_WAIT_FOR,%P 2:NOT, 4:, 5:$IN, 6:129, 7:AVA/REC MESA B, 9:
WAIT FOR  NOT ( $IN[129] )
;ENDFOLD
END

--- NEW_MASTER_MESA_A.dat ---
&ACCESS RVP
&REL 381
&PARAM EDITMASK = *
&PARAM TEMPLATE = C:\KRC\Roboter\Template\vorgabe
&PARAM DISKPATH = KRC:\R1\Program\Solda\MASTER_125
DEFDAT  NEW_MASTER_MESA_A
;FOLD EXTERNAL DECLARATIONS;%{PE}%MKUKATPBASIS,%CEXT,%VCOMMON,%P
;FOLD BASISTECH EXT;%{PE}%MKUKATPBASIS,%CEXT,%VEXT,%P
EXT  BAS (BAS_COMMAND  :IN,REAL  :IN )
DECL INT SUCCESS
;ENDFOLD (BASISTECH EXT)
;FOLD USER EXT;%{E}%MKUKATPUSER,%CEXT,%VEXT,%P
;Make your modifications here

;ENDFOLD (USER EXT)
;ENDFOLD (EXTERNAL DECLARATIONS)
DECL ATBg_Start_T AS_WDAT1={JobModeId 1306102413,ParamSetId -1047099609,StartTime 0.0,PreFlowTime 0.0,Channel1 0.0,Channel2 2.00000,Channel3 0.0,Channel4 0.0,Channel5 0.0,Channel6 0.0,Channel7 0.0,Channel8 0.0,PurgeTime 0.0}
DECL ATBg_Weld_T AW_WDAT1={JobModeId -187662529,ParamSetId -430485013,Velocity 0.00830000,Channel1 30.0000,Channel2 1.00000,Channel3 0.0,Channel4 0.0,Channel5 0.0,Channel6 0.0,Channel7 0.0,Channel8 0.0}
DECL WTCg_WeaveDefinition_T WV_WDAT1={Pattern #None,Length 4.00000,Amplitude 2.00000,Angle 0.0}
DECL FDAT FP1={TOOL_NO 1,BASE_NO 0,IPO_FRAME #BASE,POINT2[] " ",TQ_STATE FALSE}
DECL PDAT PPDAT1={ACC 100.000,APO_DIST 100.000,APO_MODE #CPTP,GEAR_JERK 50.0000}
DECL E6POS XP1={X 1496.76196,Y 582.870911,Z 1275.91040,A 159.098511,B 49.1786919,C -124.034058,S 0,T 43,E1 180.001038,E2 179.999084,E3 180.004181,E4 0.0,E5 0.0,E6 0.0}
DECL MODULEPARAM_T LAST_TP_PARAMS={PARAMS[] "Kuka.MoveDataPtpName=PDAT60; Kuka.VelocityPtp=100; Kuka.PointName=P78; Kuka.BlendingEnabled=False; Kuka.FrameData.tq_state=False; Kuka.FrameData.base_no=0; Kuka.FrameData.tool_no=1; Kuka.FrameData.ipo_frame=#BASE; Kuka.MovementDataPdat.apo_mode=#CPTP; Kuka.MovementDataPdat.apo_dist=100; Kuka.MovementData.acc=100; Kuka.MovementData.gear_jerk=50; ArcTech.WdatVarName=WDAT39; Kuka.MoveDataName=CPDAT51; Kuka.VelocityPath=0.3; Kuka.MovementData.apo_fac=50; Kuka.MovementData.apo_dist=100; Kuka.MovementData.axis_acc=100; Kuka.MovementData.axis_vel=100; Kuka.MovementData.circ_typ=#BASE; Kuka.MovementData.exax_ign=0; Kuka.MovementData.jerk_fac=50; Kuka.MovementData.ori_typ=#VAR; Kuka.FrameData.point2=                                                                                                                                                                                                "}
DECL ATBg_Crater_T AC_WDAT2={JobModeId -187662529,ParamSetId -1375177600,CraterTime 0.100000,PostflowTime 0.100000,Channel1 30.0000,Channel2 1.00000,Channel3 0.0,Channel4 0.0,Channel5 0.0,Channel6 0.0,Channel7 0.0,Channel8 0.0,BurnBackTime 0.0}
DECL FDAT FP2={TOOL_NO 1,BASE_NO 0,IPO_FRAME #BASE,POINT2[] " ",TQ_STATE FALSE}
DECL LDAT LCPDAT1={ACC 100.000,APO_DIST 100.000,APO_FAC 50.0000,AXIS_VEL 100.000,AXIS_ACC 100.000,ORI_TYP #VAR,CIRC_TYP #BASE,JERK_FAC 50.0000,GEAR_JERK 50.0000,EXAX_IGN 0}
DECL E6POS XP2={X 1500.47852,Y 573.313171,Z 1274.83447,A 158.879135,B 49.0362473,C -123.840370,S 0,T 43,E1 180.001038,E2 179.999084,E3 180.004181,E4 0.0,E5 0.0,E6 0.0}
DECL BASIS_SUGG_T LAST_BASIS={POINT1[] "P185                    ",POINT2[] "P185                    ",CP_PARAMS[] "CPDAT0                  ",PTP_PARAMS[] "PDAT137                 ",CONT[] "C_DIS                   ",CP_VEL[] "2.0                     ",PTP_VEL[] "100                     ",SYNC_PARAMS[] "SYNCDAT                 ",SPL_NAME[] "S0                      ",A_PARAMS[] "ADAT0                   "}
DECL E6POS XP3={X 1482.70276,Y 566.674377,Z 1310.22266,A 157.428940,B 50.3861160,C -125.741325,S 0,T 43,E1 180.001038,E2 179.999084,E3 180.004181,E4 0.0,E5 0.0,E6 0.0}
DECL FDAT FP3={TOOL_NO 1,BASE_NO 0,IPO_FRAME #BASE,POINT2[] " ",TQ_STATE FALSE}
DECL PDAT PPDAT2={VEL 100.000,ACC 100.000,APO_DIST 100.000,GEAR_JERK 50.0000,EXAX_IGN 3}
DECL E6POS XP4={X 1482.70276,Y 566.674377,Z 1310.22266,A 157.428940,B 50.3861160,C -125.741325,S 0,T 43,E1 180.001038,E2 179.999084,E3 180.004181,E4 0.0,E5 0.0,E6 0.0}
DECL FDAT FP4={TOOL_NO 1,BASE_NO 0,IPO_FRAME #BASE,POINT2[] " ",TQ_STATE FALSE}
DECL PDAT PPDAT3={VEL 100.000,ACC 100.000,APO_DIST 100.000,GEAR_JERK 50.0000,EXAX_IGN 3}
DECL ATBg_Start_T AS_WDAT3={JobModeId 1306102413,ParamSetId -1047099609,StartTime 0.0,PreFlowTime 0.0,Channel1 0.0,Channel2 2.00000,Channel3 0.0,Channel4 0.0,Channel5 0.0,Channel6 0.0,Channel7 0.0,Channel8 0.0,PurgeTime 0.0}
DECL ATBg_Weld_T AW_WDAT3={JobModeId -187662529,ParamSetId -430485013,Velocity 0.00830000,Channel1 30.0000,Channel2 1.00000,Channel3 0.0,Channel4 0.0,Channel5 0.0,Channel6 0.0,Channel7 0.0,Channel8 0.0}
DECL WTCg_WeaveDefinition_T WV_WDAT3={Pattern #None,Length 4.00000,Amplitude 2.00000,Angle 0.0}
DECL FDAT FP5={TOOL_NO 1,BASE_NO 0,IPO_FRAME #BASE,POINT2[] " ",TQ_STATE FALSE}
DECL PDAT PPDAT4={ACC 100.000,APO_DIST 100.000,APO_MODE #CPTP,GEAR_JERK 50.0000}
DECL E6POS XP5={X 1466.55981,Y 697.098694,Z 1383.56360,A -77.2453308,B 24.5325470,C -35.8039818,S 0,T 11,E1 180.001022,E2 179.999100,E3 180.004028,E4 0.0,E5 0.0,E6 0.0}
DECL ATBg_Crater_T AC_WDAT4={JobModeId -187662529,ParamSetId -1375177600,CraterTime 0.100000,PostflowTime 0.100000,Channel1 30.0000,Channel2 1.00000,Channel3 0.0,Channel4 0.0,Channel5 0.0,Channel6 0.0,Channel7 0.0,Channel8 0.0,BurnBackTime 0.0}
DECL FDAT FP6={TOOL_NO 1,BASE_NO 0,IPO_FRAME #BASE,POINT2[] " ",TQ_STATE FALSE}
DECL LDAT LCPDAT2={ACC 100.000,APO_DIST 100.000,APO_FAC 50.0000,AXIS_VEL 100.000,AXIS_ACC 100.000,ORI_TYP #VAR,CIRC_TYP #BASE,JERK_FAC 50.0000,GEAR_JERK 50.0000,EXAX_IGN 0}
DECL E6POS XP6={X 1461.39319,Y 705.430176,Z 1377.38342,A -77.4356918,B 24.1875134,C -37.1046600,S 2,T 11,E1 180.001022,E2 179.999100,E3 180.004028,E4 0.0,E5 0.0,E6 0.0}
DECL LDAT LCPDAT3={ACC 100.000,APO_DIST 100.000,APO_FAC 50.0000,AXIS_VEL 100.000,AXIS_ACC 100.000,ORI_TYP #VAR,CIRC_TYP #BASE,JERK_FAC 50.0000,GEAR_JERK 50.0000,EXAX_IGN 0}
DECL LDAT LCPDAT4={ACC 100.000,APO_DIST 100.000,APO_FAC 50.0000,AXIS_VEL 100.000,AXIS_ACC 100.000,ORI_TYP #VAR,CIRC_TYP #BASE,JERK_FAC 50.0000,GEAR_JERK 50.0000,EXAX_IGN 0}
DECL PDAT PPDAT5={ACC 100.000,APO_DIST 100.000,APO_MODE #CPTP,GEAR_JERK 50.0000}
DECL ATBg_Start_T AS_WDAT5={JobModeId 1306102413,ParamSetId -1047099609,StartTime 0.0,PreFlowTime 0.0,Channel1 0.0,Channel2 2.00000,Channel3 0.0,Channel4 0.0,Channel5 0.0,Channel6 0.0,Channel7 0.0,Channel8 0.0,PurgeTime 0.0}
DECL ATBg_Weld_T AW_WDAT5={JobModeId -187662529,ParamSetId -430485013,Velocity 0.00830000,Channel1 30.0000,Channel2 1.00000,Channel3 0.0,Channel4 0.0,Channel5 0.0,Channel6 0.0,Channel7 0.0,Channel8 0.0}
DECL WTCg_WeaveDefinition_T WV_WDAT5={Pattern #None,Length 4.00000,Amplitude 2.00000,Angle 0.0}
DECL FDAT FP7={TOOL_NO 1,BASE_NO 0,IPO_FRAME #BASE,POINT2[] " ",TQ_STATE FALSE}
DECL PDAT PPDAT6={ACC 100.000,APO_DIST 100.000,APO_MODE #CPTP,GEAR_JERK 50.0000}
DECL E6POS XP7={X 1484.82764,Y 693.075134,Z 1499.31616,A -23.4080772,B -53.4302559,C -46.9197922,S 2,T 43,E1 180.001022,E2 179.999100,E3 180.004028,E4 0.0,E5 0.0,E6 0.0}
DECL ATBg_Crater_T AC_WDAT6={JobModeId -187662529,ParamSetId -1375177600,CraterTime 0.100000,PostflowTime 0.100000,Channel1 30.0000,Channel2 1.00000,Channel3 0.0,Channel4 0.0,Channel5 0.0,Channel6 0.0,Channel7 0.0,Channel8 0.0,BurnBackTime 0.0}
DECL FDAT FP8={TOOL_NO 1,BASE_NO 0,IPO_FRAME #BASE,POINT2[] " ",TQ_STATE FALSE}
DECL LDAT LCPDAT5={ACC 100.000,APO_DIST 100.000,APO_FAC 50.0000,AXIS_VEL 100.000,AXIS_ACC 100.000,ORI_TYP #VAR,CIRC_TYP #BASE,JERK_FAC 50.0000,GEAR_JERK 50.0000,EXAX_IGN 0}
DECL E6POS XP8={X 1489.87585,Y 680.574158,Z 1497.46960,A -29.8228798,B -49.4180946,C -42.0220261,S 2,T 43,E1 180.001022,E2 179.999100,E3 180.004028,E4 0.0,E5 0.0,E6 0.0}
DECL E6POS XP9={X 1436.40173,Y 655.308228,Z 1566.53308,A -32.0819,B -50.6817131,C -39.0761185,S 2,T 43,E1 180.000992,E2 179.999115,E3 180.003891,E4 0.0,E5 0.0,E6 0.0}
DECL FDAT FP9={TOOL_NO 1,BASE_NO 0,IPO_FRAME #BASE,POINT2[] " ",TQ_STATE FALSE}
DECL PDAT PPDAT7={VEL 100.000,ACC 100.000,APO_DIST 100.000,GEAR_JERK 50.0000,EXAX_IGN 3}
DECL E6POS XP10={X 1436.40173,Y 655.308228,Z 1566.53308,A -32.0819,B -50.6817131,C -39.0761185,S 2,T 43,E1 180.000992,E2 179.999115,E3 180.003891,E4 0.0,E5 0.0,E6 0.0}
DECL FDAT FP10={TOOL_NO 1,BASE_NO 0,IPO_FRAME #BASE,POINT2[] " ",TQ_STATE FALSE}
DECL PDAT PPDAT8={VEL 100.000,ACC 100.000,APO_DIST 100.000,GEAR_JERK 50.0000,EXAX_IGN 3}
DECL E6POS XP11={X 963.610474,Y 468.452576,Z 2013.77759,A -55.0418549,B -77.1242065,C -9.45068359,S 2,T 43,E1 180.000992,E2 179.999115,E3 180.003891,E4 0.0,E5 0.0,E6 0.0}
DECL FDAT FP11={TOOL_NO 1,BASE_NO 0,IPO_FRAME #BASE,POINT2[] " ",TQ_STATE FALSE}
DECL PDAT PPDAT9={VEL 100.000,ACC 100.000,APO_DIST 100.000,GEAR_JERK 50.0000,EXAX_IGN 3}
DECL E6POS XP12={X 1030.98926,Y 213.392715,Z 1949.10840,A -48.0140724,B -75.1600342,C -31.3416386,S 2,T 43,E1 180.000992,E2 179.999115,E3 180.003891,E4 0.0,E5 0.0,E6 0.0}
DECL FDAT FP12={TOOL_NO 1,BASE_NO 0,IPO_FRAME #BASE,POINT2[] " ",TQ_STATE FALSE}
DECL PDAT PPDAT10={VEL 100.000,ACC 100.000,APO_DIST 100.000,GEAR_JERK 50.0000,EXAX_IGN 3}
DECL E6POS XP13={X 1582.72571,Y 214.898727,Z 1484.79297,A -17.8722897,B -60.1868629,C -67.3960724,S 2,T 43,E1 180.000992,E2 179.999115,E3 180.003891,E4 0.0,E5 0.0,E6 0.0}
DECL FDAT FP13={TOOL_NO 1,BASE_NO 0,IPO_FRAME #BASE,POINT2[] " ",TQ_STATE FALSE}
DECL PDAT PPDAT11={VEL 100.000,ACC 100.000,APO_DIST 100.000,GEAR_JERK 50.0000,EXAX_IGN 3}
DECL ATBg_Start_T AS_WDAT7={JobModeId 1306102413,ParamSetId -1047099609,StartTime 0.0,PreFlowTime 0.0,Channel1 0.0,Channel2 2.00000,Channel3 0.0,Channel4 0.0,Channel5 0.0,Channel6 0.0,Channel7 0.0,Channel8 0.0,PurgeTime 0.0}
DECL ATBg_Weld_T AW_WDAT7={JobModeId -187662529,ParamSetId -430485013,Velocity 0.00830000,Channel1 30.0000,Channel2 1.00000,Channel3 0.0,Channel4 0.0,Channel5 0.0,Channel6 0.0,Channel7 0.0,Channel8 0.0}
DECL WTCg_WeaveDefinition_T WV_WDAT7={Pattern #None,Length 4.00000,Amplitude 2.00000,Angle 0.0}
DECL FDAT FP14={TOOL_NO 1,BASE_NO 0,IPO_FRAME #BASE,POINT2[] " ",TQ_STATE FALSE}
DECL PDAT PPDAT12={ACC 100.000,APO_DIST 100.000,APO_MODE #CPTP,GEAR_JERK 50.0000}
DECL E6POS XP14={X 1584.62036,Y 215.140686,Z 1482.90674,A -17.8341675,B -60.1402512,C -67.4400177,S 2,T 43,E1 180.000992,E2 179.999115,E3 180.003891,E4 0.0,E5 0.0,E6 0.0}
DECL ATBg_Crater_T AC_WDAT8={JobModeId -187662529,ParamSetId -1375177600,CraterTime 0.100000,PostflowTime 0.100000,Channel1 30.0000,Channel2 1.00000,Channel3 0.0,Channel4 0.0,Channel5 0.0,Channel6 0.0,Channel7 0.0,Channel8 0.0,BurnBackTime 0.0}
DECL FDAT FP15={TOOL_NO 1,BASE_NO 0,IPO_FRAME #BASE,POINT2[] " ",TQ_STATE FALSE}
DECL LDAT LCPDAT6={ACC 100.000,APO_DIST 100.000,APO_FAC 50.0000,AXIS_VEL 100.000,AXIS_ACC 100.000,ORI_TYP #VAR,CIRC_TYP #BASE,JERK_FAC 50.0000,GEAR_JERK 50.0000,EXAX_IGN 0}
DECL E6POS XP15={X 1584.62036,Y 215.140686,Z 1482.90674,A -17.8341675,B -60.1402512,C -67.4400177,S 2,T 43,E1 180.000992,E2 179.999115,E3 180.003891,E4 0.0,E5 0.0,E6 0.0}
DECL E6POS XP16={X 1547.48352,Y 210.398209,Z 1520.88965,A -18.7159042,B -61.1769409,C -66.4285660,S 2,T 43,E1 180.000992,E2 179.999115,E3 180.003891,E4 0.0,E5 0.0,E6 0.0}
DECL FDAT FP16={TOOL_NO 1,BASE_NO 0,IPO_FRAME #BASE,POINT2[] " ",TQ_STATE FALSE}
DECL PDAT PPDAT13={VEL 100.000,ACC 100.000,APO_DIST 100.000,GEAR_JERK 50.0000,EXAX_IGN 3}
DECL E6POS XP17={X 1505.81213,Y 205.076660,Z 1574.12085,A -20.5965290,B -63.1322670,C -64.3020325,S 2,T 43,E1 180.000992,E2 179.999115,E3 180.003891,E4 0.0,E5 0.0,E6 0.0}
DECL FDAT FP17={TOOL_NO 1,BASE_NO 0,IPO_FRAME #BASE,POINT2[] " ",TQ_STATE FALSE}
DECL PDAT PPDAT14={VEL 100.000,ACC 100.000,APO_DIST 100.000,GEAR_JERK 50.0000,EXAX_IGN 3}
DECL E6POS XP18={X 1562.25806,Y 172.455948,Z 1399.03113,A -178.023010,B 72.2041321,C -95.4785080,S 2,T 43,E1 180.000992,E2 179.999115,E3 180.003891,E4 0.0,E5 0.0,E6 0.0}
DECL FDAT FP18={TOOL_NO 1,BASE_NO 0,IPO_FRAME #BASE,POINT2[] " ",TQ_STATE FALSE}
DECL PDAT PPDAT15={VEL 100.000,ACC 100.000,APO_DIST 100.000,GEAR_JERK 50.0000,EXAX_IGN 3}
DECL ATBg_Start_T AS_WDAT9={JobModeId 1306102413,ParamSetId -1047099609,StartTime 0.0,PreFlowTime 0.0,Channel1 0.0,Channel2 2.00000,Channel3 0.0,Channel4 0.0,Channel5 0.0,Channel6 0.0,Channel7 0.0,Channel8 0.0,PurgeTime 0.0}
DECL ATBg_Weld_T AW_WDAT9={JobModeId -187662529,ParamSetId -430485013,Velocity 0.00830000,Channel1 30.0000,Channel2 1.00000,Channel3 0.0,Channel4 0.0,Channel5 0.0,Channel6 0.0,Channel7 0.0,Channel8 0.0}
DECL WTCg_WeaveDefinition_T WV_WDAT9={Pattern #None,Length 4.00000,Amplitude 2.00000,Angle 0.0}
DECL FDAT FP19={TOOL_NO 1,BASE_NO 0,IPO_FRAME #BASE,POINT2[] " ",TQ_STATE FALSE}
DECL PDAT PPDAT16={ACC 100.000,APO_DIST 100.000,APO_MODE #CPTP,GEAR_JERK 50.0000}
DECL E6POS XP19={X 1594.61816,Y 176.588425,Z 1348.24695,A -177.500946,B 70.1884537,C -94.9270935,S 2,T 43,E1 180.000992,E2 179.999115,E3 180.003891,E4 0.0,E5 0.0,E6 0.0}
DECL ATBg_Crater_T AC_WDAT10={JobModeId -187662529,ParamSetId -1375177600,CraterTime 0.100000,PostflowTime 0.100000,Channel1 30.0000,Channel2 1.00000,Channel3 0.0,Channel4 0.0,Channel5 0.0,Channel6 0.0,Channel7 0.0,Channel8 0.0,BurnBackTime 0.0}
DECL FDAT FP20={TOOL_NO 1,BASE_NO 0,IPO_FRAME #BASE,POINT2[] " ",TQ_STATE FALSE}
DECL LDAT LCPDAT7={ACC 100.000,APO_DIST 100.000,APO_FAC 50.0000,AXIS_VEL 100.000,AXIS_ACC 100.000,ORI_TYP #VAR,CIRC_TYP #BASE,JERK_FAC 50.0000,GEAR_JERK 50.0000,EXAX_IGN 0}
DECL E6POS XP20={X 1594.61816,Y 176.588425,Z 1348.24695,A -177.500946,B 70.1884537,C -94.9270935,S 2,T 43,E1 180.000992,E2 179.999115,E3 180.003891,E4 0.0,E5 0.0,E6 0.0}
DECL E6POS XP21={X 1562.25806,Y 172.455933,Z 1399.03113,A -178.023010,B 72.2041321,C -95.4785080,S 2,T 43,E1 180.000992,E2 179.999115,E3 180.003891,E4 0.0,E5 0.0,E6 0.0}
DECL FDAT FP21={TOOL_NO 1,BASE_NO 0,IPO_FRAME #BASE,POINT2[] " ",TQ_STATE FALSE}
DECL PDAT PPDAT17={VEL 100.000,ACC 100.000,APO_DIST 100.000,GEAR_JERK 50.0000,EXAX_IGN 3}
DECL E6POS XP22={X 1528.15576,Y 167.507034,Z 1565.51379,A 28.2313652,B 85.1708,C 110.647263,S 2,T 43,E1 180.000992,E2 179.999115,E3 180.003891,E4 0.0,E5 0.0,E6 0.0}
DECL FDAT FP22={TOOL_NO 1,BASE_NO 0,IPO_FRAME #BASE,POINT2[] " ",TQ_STATE FALSE}
DECL PDAT PPDAT18={VEL 100.000,ACC 100.000,APO_DIST 100.000,GEAR_JERK 50.0000,EXAX_IGN 3}
DECL E6POS XP23={X 1502.60278,Y -324.416138,Z 1572.55701,A -74.3732529,B 79.7488556,C 26.2741585,S 2,T 10,E1 180.000992,E2 179.999115,E3 180.003891,E4 0.0,E5 0.0,E6 0.0}
DECL FDAT FP23={TOOL_NO 1,BASE_NO 0,IPO_FRAME #BASE,POINT2[] " ",TQ_STATE FALSE}
DECL PDAT PPDAT19={VEL 100.000,ACC 100.000,APO_DIST 100.000,GEAR_JERK 50.0000,EXAX_IGN 3}
DECL ATBg_Start_T AS_WDAT11={JobModeId 1306102413,ParamSetId -1047099609,StartTime 0.0,PreFlowTime 0.0,Channel1 0.0,Channel2 2.00000,Channel3 0.0,Channel4 0.0,Channel5 0.0,Channel6 0.0,Channel7 0.0,Channel8 0.0,PurgeTime 0.0}
DECL ATBg_Weld_T AW_WDAT11={JobModeId -187662529,ParamSetId -430485013,Velocity 0.00830000,Channel1 30.0000,Channel2 1.00000,Channel3 0.0,Channel4 0.0,Channel5 0.0,Channel6 0.0,Channel7 0.0,Channel8 0.0}
DECL WTCg_WeaveDefinition_T WV_WDAT11={Pattern #None,Length 4.00000,Amplitude 2.00000,Angle 0.0}
DECL FDAT FP24={TOOL_NO 1,BASE_NO 0,IPO_FRAME #BASE,POINT2[] " ",TQ_STATE FALSE}
DECL PDAT PPDAT20={ACC 100.000,APO_DIST 100.000,APO_MODE #CPTP,GEAR_JERK 50.0000}
DECL E6POS XP24={X 1574.90735,Y -337.206,Z 1350.69495,A -165.207779,B 67.7758102,C -66.7983551,S 2,T 10,E1 180.000992,E2 179.999115,E3 180.003891,E4 0.0,E5 0.0,E6 0.0}
DECL ATBg_Crater_T AC_WDAT12={JobModeId -187662529,ParamSetId -1375177600,CraterTime 0.100000,PostflowTime 0.100000,Channel1 30.0000,Channel2 1.00000,Channel3 0.0,Channel4 0.0,Channel5 0.0,Channel6 0.0,Channel7 0.0,Channel8 0.0,BurnBackTime 0.0}
DECL FDAT FP25={TOOL_NO 1,BASE_NO 0,IPO_FRAME #BASE,POINT2[] " ",TQ_STATE FALSE}
DECL LDAT LCPDAT8={ACC 100.000,APO_DIST 100.000,APO_FAC 50.0000,AXIS_VEL 100.000,AXIS_ACC 100.000,ORI_TYP #VAR,CIRC_TYP #BASE,JERK_FAC 50.0000,GEAR_JERK 50.0000,EXAX_IGN 0}
DECL E6POS XP25={X 1574.90735,Y -337.206,Z 1350.69495,A -165.207779,B 67.7758102,C -66.7983551,S 2,T 10,E1 180.000992,E2 179.999115,E3 180.003891,E4 0.0,E5 0.0,E6 0.0}
DECL E6POS XP26={X 1522.26257,Y -327.427399,Z 1432.21021,A -161.269516,B 70.6730652,C -62.5877876,S 2,T 10,E1 180.000992,E2 179.999115,E3 180.003891,E4 0.0,E5 0.0,E6 0.0}
DECL FDAT FP26={TOOL_NO 1,BASE_NO 0,IPO_FRAME #BASE,POINT2[] " ",TQ_STATE FALSE}
DECL PDAT PPDAT21={VEL 100.000,ACC 100.000,APO_DIST 100.000,GEAR_JERK 50.0000,EXAX_IGN 3}
DECL E6POS XP27={X 1491.06848,Y -228.728851,Z 1583.72083,A 11.7713518,B -64.7742691,C -109.904411,S 2,T 10,E1 180.000992,E2 179.999115,E3 180.003891,E4 0.0,E5 0.0,E6 0.0}
DECL FDAT FP27={TOOL_NO 1,BASE_NO 0,IPO_FRAME #BASE,POINT2[] " ",TQ_STATE FALSE}
DECL PDAT PPDAT22={VEL 100.000,ACC 100.000,APO_DIST 100.000,GEAR_JERK 50.0000,EXAX_IGN 3}
DECL ATBg_Start_T AS_WDAT13={JobModeId 1306102413,ParamSetId -1047099609,StartTime 0.0,PreFlowTime 0.0,Channel1 0.0,Channel2 2.00000,Channel3 0.0,Channel4 0.0,Channel5 0.0,Channel6 0.0,Channel7 0.0,Channel8 0.0,PurgeTime 0.0}
DECL ATBg_Weld_T AW_WDAT13={JobModeId -187662529,ParamSetId -430485013,Velocity 0.00830000,Channel1 30.0000,Channel2 1.00000,Channel3 0.0,Channel4 0.0,Channel5 0.0,Channel6 0.0,Channel7 0.0,Channel8 0.0}
DECL WTCg_WeaveDefinition_T WV_WDAT13={Pattern #None,Length 4.00000,Amplitude 2.00000,Angle 0.0}
DECL FDAT FP28={TOOL_NO 1,BASE_NO 0,IPO_FRAME #BASE,POINT2[] " ",TQ_STATE FALSE}
DECL PDAT PPDAT23={ACC 100.000,APO_DIST 100.000,APO_MODE #CPTP,GEAR_JERK 50.0000}
DECL E6POS XP28={X 1572.85193,Y -243.939880,Z 1478.24158,A 8.99041462,B -61.0612869,C -106.788139,S 2,T 10,E1 180.000992,E2 179.999115,E3 180.003891,E4 0.0,E5 0.0,E6 0.0}
DECL ATBg_Crater_T AC_WDAT14={JobModeId -187662529,ParamSetId -1375177600,CraterTime 0.100000,PostflowTime 0.100000,Channel1 30.0000,Channel2 1.00000,Channel3 0.0,Channel4 0.0,Channel5 0.0,Channel6 0.0,Channel7 0.0,Channel8 0.0,BurnBackTime 0.0}
DECL FDAT FP29={TOOL_NO 1,BASE_NO 0,IPO_FRAME #BASE,POINT2[] " ",TQ_STATE FALSE}
DECL LDAT LCPDAT9={ACC 100.000,APO_DIST 100.000,APO_FAC 50.0000,AXIS_VEL 100.000,AXIS_ACC 100.000,ORI_TYP #VAR,CIRC_TYP #BASE,JERK_FAC 50.0000,GEAR_JERK 50.0000,EXAX_IGN 0}
DECL E6POS XP29={X 1572.85193,Y -243.939880,Z 1478.24158,A 8.99041462,B -61.0612869,C -106.788139,S 2,T 10,E1 180.000992,E2 179.999115,E3 180.003891,E4 0.0,E5 0.0,E6 0.0}
DECL E6POS XP30={X 1435.31335,Y -218.392578,Z 1621.85400,A 12.7399940,B -65.8434830,C -110.975647,S 2,T 10,E1 180.000992,E2 179.999115,E3 180.003891,E4 0.0,E5 0.0,E6 0.0}
DECL FDAT FP30={TOOL_NO 1,BASE_NO 0,IPO_FRAME #BASE,POINT2[] " ",TQ_STATE FALSE}
DECL PDAT PPDAT24={VEL 100.000,ACC 100.000,APO_DIST 100.000,GEAR_JERK 50.0000,EXAX_IGN 3}
DECL E6POS XP31={X 1211.71753,Y -176.207092,Z 1775.64709,A 10.2153435,B -62.4659920,C -107.999146,S 2,T 10,E1 180.000992,E2 179.999115,E3 180.003891,E4 0.0,E5 0.0,E6 0.0}
DECL FDAT FP31={TOOL_NO 1,BASE_NO 0,IPO_FRAME #BASE,POINT2[] " ",TQ_STATE FALSE}
DECL PDAT PPDAT25={VEL 100.000,ACC 100.000,APO_DIST 100.000,GEAR_JERK 50.0000,EXAX_IGN 3}
DECL E6POS XP32={X 1115.09851,Y -492.561127,Z 1780.23438,A 33.0263557,B -54.0004311,C -144.370392,S 2,T 10,E1 180.000992,E2 179.999115,E3 180.003891,E4 0.0,E5 0.0,E6 0.0}
DECL FDAT FP32={TOOL_NO 1,BASE_NO 0,IPO_FRAME #BASE,POINT2[] " ",TQ_STATE FALSE}
DECL PDAT PPDAT26={VEL 100.000,ACC 100.000,APO_DIST 100.000,GEAR_JERK 50.0000,EXAX_IGN 3}
DECL ATBg_Start_T AS_WDAT15={JobModeId 1306102413,ParamSetId -1047099609,StartTime 0.0,PreFlowTime 0.0,Channel1 0.0,Channel2 2.00000,Channel3 0.0,Channel4 0.0,Channel5 0.0,Channel6 0.0,Channel7 0.0,Channel8 0.0,PurgeTime 0.0}
DECL ATBg_Weld_T AW_WDAT15={JobModeId -187662529,ParamSetId -430485013,Velocity 0.00830000,Channel1 30.0000,Channel2 1.00000,Channel3 0.0,Channel4 0.0,Channel5 0.0,Channel6 0.0,Channel7 0.0,Channel8 0.0}
DECL WTCg_WeaveDefinition_T WV_WDAT15={Pattern #None,Length 4.00000,Amplitude 2.00000,Angle 0.0}
DECL FDAT FP33={TOOL_NO 1,BASE_NO 0,IPO_FRAME #BASE,POINT2[] " ",TQ_STATE FALSE}
DECL PDAT PPDAT27={ACC 100.000,APO_DIST 100.000,APO_MODE #CPTP,GEAR_JERK 50.0000}
DECL E6POS XP33={X 1497.54565,Y -521.613,Z 1444.21875,A 57.3688469,B 47.0705,C 163.948288,S 6,T 58,E1 180.000992,E2 179.999115,E3 180.003891,E4 0.0,E5 0.0,E6 0.0}
DECL ATBg_Crater_T AC_WDAT16={JobModeId -187662529,ParamSetId -1375177600,CraterTime 0.100000,PostflowTime 0.100000,Channel1 30.0000,Channel2 1.00000,Channel3 0.0,Channel4 0.0,Channel5 0.0,Channel6 0.0,Channel7 0.0,Channel8 0.0,BurnBackTime 0.0}
DECL FDAT FP34={TOOL_NO 1,BASE_NO 0,IPO_FRAME #BASE,POINT2[] " ",TQ_STATE FALSE}
DECL LDAT LCPDAT10={ACC 100.000,APO_DIST 100.000,APO_FAC 50.0000,AXIS_VEL 100.000,AXIS_ACC 100.000,ORI_TYP #VAR,CIRC_TYP #BASE,JERK_FAC 50.0000,GEAR_JERK 50.0000,EXAX_IGN 0}
DECL E6POS XP34={X 1497.54565,Y -521.613,Z 1444.21875,A 57.3688469,B 47.0705,C 163.948288,S 6,T 58,E1 180.000992,E2 179.999115,E3 180.003891,E4 0.0,E5 0.0,E6 0.0}
DECL ATBg_Start_T AS_WDAT17={JobModeId 1306102413,ParamSetId -1047099609,StartTime 0.0,PreFlowTime 0.0,Channel1 0.0,Channel2 2.00000,Channel3 0.0,Channel4 0.0,Channel5 0.0,Channel6 0.0,Channel7 0.0,Channel8 0.0,PurgeTime 0.0}
DECL ATBg_Weld_T AW_WDAT17={JobModeId -187662529,ParamSetId -430485013,Velocity 0.00830000,Channel1 30.0000,Channel2 1.00000,Channel3 0.0,Channel4 0.0,Channel5 0.0,Channel6 0.0,Channel7 0.0,Channel8 0.0}
DECL WTCg_WeaveDefinition_T WV_WDAT17={Pattern #None,Length 4.00000,Amplitude 2.00000,Angle 0.0}
DECL FDAT FP35={TOOL_NO 1,BASE_NO 0,IPO_FRAME #BASE,POINT2[] " ",TQ_STATE FALSE}
DECL PDAT PPDAT28={ACC 100.000,APO_DIST 100.000,APO_MODE #CPTP,GEAR_JERK 50.0000}
DECL E6POS XP35={X 1490.85339,Y -544.309875,Z 1445.73792,A 56.1921425,B 47.0849609,C 163.538742,S 6,T 58,E1 180.000992,E2 179.999115,E3 180.003891,E4 0.0,E5 0.0,E6 0.0}
DECL ATBg_Crater_T AC_WDAT18={JobModeId -187662529,ParamSetId -1375177600,CraterTime 0.100000,PostflowTime 0.100000,Channel1 30.0000,Channel2 1.00000,Channel3 0.0,Channel4 0.0,Channel5 0.0,Channel6 0.0,Channel7 0.0,Channel8 0.0,BurnBackTime 0.0}
DECL FDAT FP36={TOOL_NO 1,BASE_NO 0,IPO_FRAME #BASE,POINT2[] " ",TQ_STATE FALSE}
DECL LDAT LCPDAT11={ACC 100.000,APO_DIST 100.000,APO_FAC 50.0000,AXIS_VEL 100.000,AXIS_ACC 100.000,ORI_TYP #VAR,CIRC_TYP #BASE,JERK_FAC 50.0000,GEAR_JERK 50.0000,EXAX_IGN 0}
DECL E6POS XP36={X 1490.85339,Y -544.309875,Z 1445.73792,A 56.1921425,B 47.0849609,C 163.538742,S 6,T 58,E1 180.000992,E2 179.999115,E3 180.003891,E4 0.0,E5 0.0,E6 0.0}
DECL ATBg_Start_T AS_WDAT19={JobModeId 1306102413,ParamSetId -1047099609,StartTime 0.0,PreFlowTime 0.0,Channel1 0.0,Channel2 2.00000,Channel3 0.0,Channel4 0.0,Channel5 0.0,Channel6 0.0,Channel7 0.0,Channel8 0.0,PurgeTime 0.0}
DECL ATBg_Weld_T AW_WDAT19={JobModeId -187662529,ParamSetId -430485013,Velocity 0.00830000,Channel1 30.0000,Channel2 1.00000,Channel3 0.0,Channel4 0.0,Channel5 0.0,Channel6 0.0,Channel7 0.0,Channel8 0.0}
DECL WTCg_WeaveDefinition_T WV_WDAT19={Pattern #None,Length 4.00000,Amplitude 2.00000,Angle 0.0}
DECL FDAT FP37={TOOL_NO 1,BASE_NO 0,IPO_FRAME #BASE,POINT2[] " ",TQ_STATE FALSE}
DECL PDAT PPDAT29={ACC 100.000,APO_DIST 100.000,APO_MODE #CPTP,GEAR_JERK 50.0000}
DECL E6POS XP37={X 1451.87244,Y -698.568726,Z 1532.68176,A -109.570,B -5.58304501,C 1.80761051,S 2,T 42,E1 180.000992,E2 179.999115,E3 180.003891,E4 0.0,E5 0.0,E6 0.0}
DECL ATBg_Crater_T AC_WDAT20={JobModeId -187662529,ParamSetId -1375177600,CraterTime 0.100000,PostflowTime 0.100000,Channel1 30.0000,Channel2 1.00000,Channel3 0.0,Channel4 0.0,Channel5 0.0,Channel6 0.0,Channel7 0.0,Channel8 0.0,BurnBackTime 0.0}
DECL FDAT FP38={TOOL_NO 1,BASE_NO 0,IPO_FRAME #BASE,POINT2[] " ",TQ_STATE FALSE}
DECL LDAT LCPDAT12={ACC 100.000,APO_DIST 100.000,APO_FAC 50.0000,AXIS_VEL 100.000,AXIS_ACC 100.000,ORI_TYP #VAR,CIRC_TYP #BASE,JERK_FAC 50.0000,GEAR_JERK 50.0000,EXAX_IGN 0}
DECL E6POS XP38={X 1451.87244,Y -698.568726,Z 1532.68176,A -109.570,B -5.58304501,C 1.80761051,S 2,T 42,E1 180.000992,E2 179.999115,E3 180.003891,E4 0.0,E5 0.0,E6 0.0}
DECL ATBg_Start_T AS_WDAT21={JobModeId 1306102413,ParamSetId -1047099609,StartTime 0.0,PreFlowTime 0.0,Channel1 0.0,Channel2 2.00000,Channel3 0.0,Channel4 0.0,Channel5 0.0,Channel6 0.0,Channel7 0.0,Channel8 0.0,PurgeTime 0.0}
DECL ATBg_Weld_T AW_WDAT21={JobModeId -187662529,ParamSetId -430485013,Velocity 0.00830000,Channel1 30.0000,Channel2 1.00000,Channel3 0.0,Channel4 0.0,Channel5 0.0,Channel6 0.0,Channel7 0.0,Channel8 0.0}
DECL WTCg_WeaveDefinition_T WV_WDAT21={Pattern #None,Length 4.00000,Amplitude 2.00000,Angle 0.0}
DECL FDAT FP39={TOOL_NO 1,BASE_NO 0,IPO_FRAME #BASE,POINT2[] " ",TQ_STATE FALSE}
DECL PDAT PPDAT30={ACC 100.000,APO_DIST 100.000,APO_MODE #CPTP,GEAR_JERK 50.0000}
DECL E6POS XP39={X 1465.31274,Y -658.103333,Z 1529.15979,A -108.004921,B -5.55257273,C 1.30878568,S 2,T 42,E1 180.000992,E2 179.999115,E3 180.003891,E4 0.0,E5 0.0,E6 0.0}
DECL ATBg_Crater_T AC_WDAT22={JobModeId -187662529,ParamSetId -1375177600,CraterTime 0.100000,PostflowTime 0.100000,Channel1 30.0000,Channel2 1.00000,Channel3 0.0,Channel4 0.0,Channel5 0.0,Channel6 0.0,Channel7 0.0,Channel8 0.0,BurnBackTime 0.0}
DECL FDAT FP40={TOOL_NO 1,BASE_NO 0,IPO_FRAME #BASE,POINT2[] " ",TQ_STATE FALSE}
DECL LDAT LCPDAT13={ACC 100.000,APO_DIST 100.000,APO_FAC 50.0000,AXIS_VEL 100.000,AXIS_ACC 100.000,ORI_TYP #VAR,CIRC_TYP #BASE,JERK_FAC 50.0000,GEAR_JERK 50.0000,EXAX_IGN 0}
DECL E6POS XP40={X 1465.31274,Y -658.103333,Z 1529.15979,A -108.004921,B -5.55257273,C 1.30878568,S 2,T 42,E1 180.000992,E2 179.999115,E3 180.003891,E4 0.0,E5 0.0,E6 0.0}
DECL E6POS XP41={X 1407.73132,Y -635.373413,Z 1607.95020,A -108.317863,B -5.73952579,C 4.48886776,S 2,T 42,E1 180.000992,E2 179.999115,E3 180.003891,E4 0.0,E5 0.0,E6 0.0}
DECL FDAT FP41={TOOL_NO 1,BASE_NO 0,IPO_FRAME #BASE,POINT2[] " ",TQ_STATE FALSE}
DECL PDAT PPDAT31={VEL 100.000,ACC 100.000,APO_DIST 100.000,GEAR_JERK 50.0000,EXAX_IGN 3}
DECL E6POS XP42={X 1421.12781,Y -644.572815,Z 1538.56335,A -91.9589157,B 50.3912086,C 18.5021782,S 2,T 42,E1 180.000992,E2 179.999115,E3 180.003891,E4 0.0,E5 0.0,E6 0.0}
DECL FDAT FP42={TOOL_NO 1,BASE_NO 0,IPO_FRAME #BASE,POINT2[] " ",TQ_STATE FALSE}
DECL PDAT PPDAT32={VEL 100.000,ACC 100.000,APO_DIST 100.000,GEAR_JERK 50.0000,EXAX_IGN 3}
DECL ATBg_Start_T AS_WDAT23={JobModeId 1306102413,ParamSetId -1047099609,StartTime 0.0,PreFlowTime 0.0,Channel1 0.0,Channel2 2.00000,Channel3 0.0,Channel4 0.0,Channel5 0.0,Channel6 0.0,Channel7 0.0,Channel8 0.0,PurgeTime 0.0}
DECL ATBg_Weld_T AW_WDAT23={JobModeId -187662529,ParamSetId -430485013,Velocity 0.00830000,Channel1 30.0000,Channel2 1.00000,Channel3 0.0,Channel4 0.0,Channel5 0.0,Channel6 0.0,Channel7 0.0,Channel8 0.0}
DECL WTCg_WeaveDefinition_T WV_WDAT23={Pattern #None,Length 4.00000,Amplitude 2.00000,Angle 0.0}
DECL FDAT FP43={TOOL_NO 1,BASE_NO 0,IPO_FRAME #BASE,POINT2[] " ",TQ_STATE FALSE}
DECL PDAT PPDAT33={ACC 100.000,APO_DIST 100.000,APO_MODE #CPTP,GEAR_JERK 50.0000}
DECL E6POS XP43={X 1502.02258,Y -578.292908,Z 1485.39441,A 30.5960255,B -59.1033821,C -140.023438,S 2,T 34,E1 180.000992,E2 179.999115,E3 180.003891,E4 0.0,E5 0.0,E6 0.0}
DECL ATBg_Crater_T AC_WDAT24={JobModeId -187662529,ParamSetId -1375177600,CraterTime 0.100000,PostflowTime 0.100000,Channel1 30.0000,Channel2 1.00000,Channel3 0.0,Channel4 0.0,Channel5 0.0,Channel6 0.0,Channel7 0.0,Channel8 0.0,BurnBackTime 0.0}
DECL FDAT FP44={TOOL_NO 1,BASE_NO 0,IPO_FRAME #BASE,POINT2[] " ",TQ_STATE FALSE}
DECL LDAT LCPDAT14={ACC 100.000,APO_DIST 100.000,APO_FAC 50.0000,AXIS_VEL 100.000,AXIS_ACC 100.000,ORI_TYP #VAR,CIRC_TYP #BASE,JERK_FAC 50.0000,GEAR_JERK 50.0000,EXAX_IGN 0}
DECL E6POS XP44={X 1502.02258,Y -578.292908,Z 1485.39441,A 30.5960255,B -59.1033821,C -140.023438,S 2,T 34,E1 180.000992,E2 179.999115,E3 180.003891,E4 0.0,E5 0.0,E6 0.0}
DECL E6POS XP45={X 1469.80408,Y -564.354736,Z 1523.67297,A 32.2780914,B -59.8028679,C -141.976486,S 2,T 34,E1 180.000992,E2 179.999115,E3 180.003891,E4 0.0,E5 0.0,E6 0.0}
DECL FDAT FP45={TOOL_NO 1,BASE_NO 0,IPO_FRAME #BASE,POINT2[] " ",TQ_STATE FALSE}
DECL PDAT PPDAT34={VEL 100.000,ACC 100.000,APO_DIST 100.000,GEAR_JERK 50.0000,EXAX_IGN 3}
DECL E6POS XP46={X 1469.80408,Y -564.354736,Z 1523.67297,A 32.2780914,B -59.8028679,C -141.976486,S 2,T 34,E1 180.000992,E2 179.999115,E3 180.003891,E4 0.0,E5 0.0,E6 0.0}
DECL FDAT FP46={TOOL_NO 1,BASE_NO 0,IPO_FRAME #BASE,POINT2[] " ",TQ_STATE FALSE}
DECL PDAT PPDAT35={VEL 100.000,ACC 100.000,APO_DIST 100.000,GEAR_JERK 50.0000,EXAX_IGN 3}
DECL ATBg_Start_T AS_WDAT25={JobModeId 1306102413,ParamSetId -1047099609,StartTime 0.0,PreFlowTime 0.0,Channel1 0.0,Channel2 2.00000,Channel3 0.0,Channel4 0.0,Channel5 0.0,Channel6 0.0,Channel7 0.0,Channel8 0.0,PurgeTime 0.0}
DECL ATBg_Weld_T AW_WDAT25={JobModeId -187662529,ParamSetId -430485013,Velocity 0.00830000,Channel1 30.0000,Channel2 1.00000,Channel3 0.0,Channel4 0.0,Channel5 0.0,Channel6 0.0,Channel7 0.0,Channel8 0.0}
DECL WTCg_WeaveDefinition_T WV_WDAT25={Pattern #None,Length 4.00000,Amplitude 2.00000,Angle 0.0}
DECL FDAT FP47={TOOL_NO 1,BASE_NO 0,IPO_FRAME #BASE,POINT2[] " ",TQ_STATE FALSE}
DECL PDAT PPDAT36={ACC 100.000,APO_DIST 100.000,APO_MODE #CPTP,GEAR_JERK 50.0000}
DECL E6POS XP47={X 1496.14221,Y -641.526245,Z 1369.59412,A -162.322510,B 68.5570297,C -52.6379738,S 2,T 2,E1 180.000992,E2 179.999115,E3 180.003891,E4 0.0,E5 0.0,E6 0.0}
DECL ATBg_Crater_T AC_WDAT26={JobModeId -187662529,ParamSetId -1375177600,CraterTime 0.100000,PostflowTime 0.100000,Channel1 30.0000,Channel2 1.00000,Channel3 0.0,Channel4 0.0,Channel5 0.0,Channel6 0.0,Channel7 0.0,Channel8 0.0,BurnBackTime 0.0}
DECL FDAT FP48={TOOL_NO 1,BASE_NO 0,IPO_FRAME #BASE,POINT2[] " ",TQ_STATE FALSE}
DECL LDAT LCPDAT15={ACC 100.000,APO_DIST 100.000,APO_FAC 50.0000,AXIS_VEL 100.000,AXIS_ACC 100.000,ORI_TYP #VAR,CIRC_TYP #BASE,JERK_FAC 50.0000,GEAR_JERK 50.0000,EXAX_IGN 0}
DECL E6POS XP48={X 1496.14221,Y -641.526245,Z 1369.59412,A -162.322510,B 68.5570297,C -52.6379738,S 2,T 2,E1 180.000992,E2 179.999115,E3 180.003891,E4 0.0,E5 0.0,E6 0.0}
DECL E6POS XP49={X 1448.11340,Y -622.753418,Z 1447.66052,A -156.764099,B 70.8568649,C -46.7135544,S 2,T 2,E1 180.000992,E2 179.999115,E3 180.003891,E4 0.0,E5 0.0,E6 0.0}
DECL FDAT FP49={TOOL_NO 1,BASE_NO 0,IPO_FRAME #BASE,POINT2[] " ",TQ_STATE FALSE}
DECL PDAT PPDAT37={VEL 100.000,ACC 100.000,APO_DIST 100.000,GEAR_JERK 50.0000,EXAX_IGN 3}
DECL E6POS XP50={X 1448.11340,Y -622.753418,Z 1447.66052,A -156.764099,B 70.8568649,C -46.7135544,S 2,T 2,E1 180.000992,E2 179.999115,E3 180.003891,E4 0.0,E5 0.0,E6 0.0}
DECL FDAT FP50={TOOL_NO 1,BASE_NO 0,IPO_FRAME #BASE,POINT2[] " ",TQ_STATE FALSE}
DECL PDAT PPDAT38={VEL 100.000,ACC 100.000,APO_DIST 100.000,GEAR_JERK 50.0000,EXAX_IGN 3}
DECL E6POS XP51={X 1485.35083,Y -636.504089,Z 1557.27551,A -66.0490341,B 70.7464371,C 47.0452,S 2,T 2,E1 180.000992,E2 179.999115,E3 180.003891,E4 0.0,E5 0.0,E6 0.0}
DECL FDAT FP51={TOOL_NO 1,BASE_NO 0,IPO_FRAME #BASE,POINT2[] " ",TQ_STATE FALSE}
DECL PDAT PPDAT39={VEL 100.000,ACC 100.000,APO_DIST 100.000,GEAR_JERK 50.0000,EXAX_IGN 3}
DECL ATBg_Start_T AS_WDAT27={JobModeId 1306102413,ParamSetId -1047099609,StartTime 0.0,PreFlowTime 0.0,Channel1 0.0,Channel2 2.00000,Channel3 0.0,Channel4 0.0,Channel5 0.0,Channel6 0.0,Channel7 0.0,Channel8 0.0,PurgeTime 0.0}
DECL ATBg_Weld_T AW_WDAT27={JobModeId -187662529,ParamSetId -430485013,Velocity 0.00830000,Channel1 30.0000,Channel2 1.00000,Channel3 0.0,Channel4 0.0,Channel5 0.0,Channel6 0.0,Channel7 0.0,Channel8 0.0}
DECL WTCg_WeaveDefinition_T WV_WDAT27={Pattern #None,Length 4.00000,Amplitude 2.00000,Angle 0.0}
DECL FDAT FP52={TOOL_NO 1,BASE_NO 0,IPO_FRAME #BASE,POINT2[] " ",TQ_STATE FALSE}
DECL PDAT PPDAT40={ACC 100.000,APO_DIST 100.000,APO_MODE #CPTP,GEAR_JERK 50.0000}
DECL E6POS XP52={X 1397.64026,Y -887.686279,Z 1403.38208,A -132.315063,B 46.3046303,C -23.7647057,S 2,T 10,E1 180.000992,E2 179.999115,E3 180.003891,E4 0.0,E5 0.0,E6 0.0}
DECL ATBg_Crater_T AC_WDAT28={JobModeId -187662529,ParamSetId -1375177600,CraterTime 0.100000,PostflowTime 0.100000,Channel1 30.0000,Channel2 1.00000,Channel3 0.0,Channel4 0.0,Channel5 0.0,Channel6 0.0,Channel7 0.0,Channel8 0.0,BurnBackTime 0.0}
DECL FDAT FP53={TOOL_NO 1,BASE_NO 0,IPO_FRAME #BASE,POINT2[] " ",TQ_STATE FALSE}
DECL LDAT LCPDAT16={ACC 100.000,APO_DIST 100.000,APO_FAC 50.0000,AXIS_VEL 100.000,AXIS_ACC 100.000,ORI_TYP #VAR,CIRC_TYP #BASE,JERK_FAC 50.0000,GEAR_JERK 50.0000,EXAX_IGN 0}
DECL E6POS XP53={X 1397.64026,Y -887.686279,Z 1403.38208,A -132.315063,B 46.3046303,C -23.7647057,S 2,T 10,E1 180.000992,E2 179.999115,E3 180.003891,E4 0.0,E5 0.0,E6 0.0}
DECL E6POS XP54={X 1367.67041,Y -870.237061,Z 1466.93665,A -128.024780,B 47.0159798,C -17.8683281,S 0,T 10,E1 180.000992,E2 179.999115,E3 180.003891,E4 0.0,E5 0.0,E6 0.0}
DECL FDAT FP54={TOOL_NO 1,BASE_NO 0,IPO_FRAME #BASE,POINT2[] " ",TQ_STATE FALSE}
DECL PDAT PPDAT41={VEL 100.000,ACC 100.000,APO_DIST 100.000,GEAR_JERK 50.0000,EXAX_IGN 3}
DECL ATBg_Start_T AS_WDAT29={JobModeId 1306102413,ParamSetId -1047099609,StartTime 0.0,PreFlowTime 0.0,Channel1 0.0,Channel2 2.00000,Channel3 0.0,Channel4 0.0,Channel5 0.0,Channel6 0.0,Channel7 0.0,Channel8 0.0,PurgeTime 0.0}
DECL ATBg_Weld_T AW_WDAT29={JobModeId -187662529,ParamSetId -430485013,Velocity 0.00830000,Channel1 30.0000,Channel2 1.00000,Channel3 0.0,Channel4 0.0,Channel5 0.0,Channel6 0.0,Channel7 0.0,Channel8 0.0}
DECL WTCg_WeaveDefinition_T WV_WDAT29={Pattern #None,Length 4.00000,Amplitude 2.00000,Angle 0.0}
DECL FDAT FP55={TOOL_NO 1,BASE_NO 0,IPO_FRAME #BASE,POINT2[] " ",TQ_STATE FALSE}
DECL PDAT PPDAT42={ACC 100.000,APO_DIST 100.000,APO_MODE #CPTP,GEAR_JERK 50.0000}
DECL E6POS XP55={X 1401.66064,Y -880.717651,Z 1461.76392,A 27.0726395,B -50.4124107,C -139.649567,S 2,T 42,E1 180.000992,E2 179.999115,E3 180.003891,E4 0.0,E5 0.0,E6 0.0}
DECL ATBg_Crater_T AC_WDAT30={JobModeId -187662529,ParamSetId -1375177600,CraterTime 0.100000,PostflowTime 0.100000,Channel1 30.0000,Channel2 1.00000,Channel3 0.0,Channel4 0.0,Channel5 0.0,Channel6 0.0,Channel7 0.0,Channel8 0.0,BurnBackTime 0.0}
DECL FDAT FP56={TOOL_NO 1,BASE_NO 0,IPO_FRAME #BASE,POINT2[] " ",TQ_STATE FALSE}
DECL LDAT LCPDAT17={ACC 100.000,APO_DIST 100.000,APO_FAC 50.0000,AXIS_VEL 100.000,AXIS_ACC 100.000,ORI_TYP #VAR,CIRC_TYP #BASE,JERK_FAC 50.0000,GEAR_JERK 50.0000,EXAX_IGN 0}
DECL E6POS XP56={X 1401.66064,Y -880.717651,Z 1461.76392,A 27.0726395,B -50.4124107,C -139.649567,S 2,T 42,E1 180.000992,E2 179.999115,E3 180.003891,E4 0.0,E5 0.0,E6 0.0}
DECL E6POS XP57={X 1369.23242,Y -857.527100,Z 1510.72119,A 28.6490726,B -51.0569115,C -141.685608,S 2,T 42,E1 180.000992,E2 179.999115,E3 180.003891,E4 0.0,E5 0.0,E6 0.0}
DECL FDAT FP57={TOOL_NO 1,BASE_NO 0,IPO_FRAME #BASE,POINT2[] " ",TQ_STATE FALSE}
DECL PDAT PPDAT43={VEL 100.000,ACC 100.000,APO_DIST 100.000,GEAR_JERK 50.0000,EXAX_IGN 3}
DECL E6POS XP58={X 1367.67041,Y -870.237061,Z 1466.93665,A -128.024780,B 47.0159798,C -17.8683281,S 0,T 10,E1 180.000992,E2 179.999115,E3 180.003891,E4 0.0,E5 0.0,E6 0.0}
DECL FDAT FP58={TOOL_NO 1,BASE_NO 0,IPO_FRAME #BASE,POINT2[] " ",TQ_STATE FALSE}
DECL PDAT PPDAT44={VEL 100.000,ACC 100.000,APO_DIST 100.000,GEAR_JERK 50.0000,EXAX_IGN 3}
DECL E6POS XP59={X 1369.23242,Y -857.527161,Z 1510.72119,A 28.6490707,B -51.0569115,C -141.685608,S 2,T 42,E1 180.000992,E2 179.999115,E3 180.003891,E4 0.0,E5 0.0,E6 0.0}
DECL FDAT FP59={TOOL_NO 1,BASE_NO 0,IPO_FRAME #BASE,POINT2[] " ",TQ_STATE FALSE}
DECL PDAT PPDAT45={VEL 100.000,ACC 100.000,APO_DIST 100.000,GEAR_JERK 50.0000,EXAX_IGN 3}
DECL E6POS XP60={X 945.867493,Y -554.763306,Z 2002.88318,A 61.1196899,B -55.2592354,C 178.350220,S 2,T 42,E1 67.5795670,E2 179.999115,E3 180.003891,E4 0.0,E5 0.0,E6 0.0}
DECL FDAT FP60={TOOL_NO 1,BASE_NO 0,IPO_FRAME #BASE,POINT2[] " ",TQ_STATE FALSE}
DECL PDAT PPDAT46={VEL 100.000,ACC 100.000,APO_DIST 100.000,GEAR_JERK 50.0000,EXAX_IGN 3}
DECL ATBg_Start_T AS_WDAT31={JobModeId 1306102413,ParamSetId -1047099609,StartTime 0.0,PreFlowTime 0.0,Channel1 0.0,Channel2 2.00000,Channel3 0.0,Channel4 0.0,Channel5 0.0,Channel6 0.0,Channel7 0.0,Channel8 0.0,PurgeTime 0.0}
DECL ATBg_Weld_T AW_WDAT31={JobModeId -187662529,ParamSetId -430485013,Velocity 0.00830000,Channel1 30.0000,Channel2 1.00000,Channel3 0.0,Channel4 0.0,Channel5 0.0,Channel6 0.0,Channel7 0.0,Channel8 0.0}
DECL WTCg_WeaveDefinition_T WV_WDAT31={Pattern #None,Length 4.00000,Amplitude 2.00000,Angle 0.0}
DECL FDAT FP61={TOOL_NO 1,BASE_NO 0,IPO_FRAME #BASE,POINT2[] " ",TQ_STATE FALSE}
DECL PDAT PPDAT47={ACC 100.000,APO_DIST 100.000,APO_MODE #CPTP,GEAR_JERK 50.0000}
DECL E6POS XP61={X 1418.66992,Y -837.542297,Z 1423.39563,A 44.6811409,B 77.4539,C 162.367722,S 2,T 42,E1 43.6475182,E2 179.999115,E3 180.003891,E4 0.0,E5 0.0,E6 0.0}
DECL ATBg_Crater_T AC_WDAT32={JobModeId -187662529,ParamSetId -1375177600,CraterTime 0.100000,PostflowTime 0.100000,Channel1 30.0000,Channel2 1.00000,Channel3 0.0,Channel4 0.0,Channel5 0.0,Channel6 0.0,Channel7 0.0,Channel8 0.0,BurnBackTime 0.0}
DECL FDAT FP62={TOOL_NO 1,BASE_NO 0,IPO_FRAME #BASE,POINT2[] " ",TQ_STATE FALSE}
DECL LDAT LCPDAT18={ACC 100.000,APO_DIST 100.000,APO_FAC 50.0000,AXIS_VEL 100.000,AXIS_ACC 100.000,ORI_TYP #VAR,CIRC_TYP #BASE,JERK_FAC 50.0000,GEAR_JERK 50.0000,EXAX_IGN 0}
DECL E6POS XP62={X 1418.66992,Y -837.542297,Z 1423.39563,A 44.6811409,B 77.4539,C 162.367722,S 2,T 42,E1 43.6475182,E2 179.999115,E3 180.003891,E4 0.0,E5 0.0,E6 0.0}
DECL E6POS XP63={X 1393.08484,Y -828.918091,Z 1461.18823,A 38.6596642,B 77.0320206,C 156.395554,S 2,T 42,E1 43.6475182,E2 179.999115,E3 180.003891,E4 0.0,E5 0.0,E6 0.0}
DECL FDAT FP63={TOOL_NO 1,BASE_NO 0,IPO_FRAME #BASE,POINT2[] " ",TQ_STATE FALSE}
DECL PDAT PPDAT48={VEL 100.000,ACC 100.000,APO_DIST 100.000,GEAR_JERK 50.0000,EXAX_IGN 3}
DECL E6POS XP64={X 1391.40466,Y -519.759521,Z 1528.67529,A 54.1671753,B 77.4182434,C 161.760574,S 2,T 42,E1 43.6475182,E2 179.999115,E3 180.003891,E4 0.0,E5 0.0,E6 0.0}
DECL FDAT FP64={TOOL_NO 1,BASE_NO 0,IPO_FRAME #BASE,POINT2[] " ",TQ_STATE FALSE}
DECL PDAT PPDAT49={VEL 100.000,ACC 100.000,APO_DIST 100.000,GEAR_JERK 50.0000,EXAX_IGN 3}
DECL E6POS XP65={X 1393.08484,Y -828.918091,Z 1461.18823,A 38.6596718,B 77.0320206,C 156.395554,S 2,T 42,E1 43.6475182,E2 179.999115,E3 180.003891,E4 0.0,E5 0.0,E6 0.0}
DECL FDAT FP65={TOOL_NO 1,BASE_NO 0,IPO_FRAME #BASE,POINT2[] " ",TQ_STATE FALSE}
DECL PDAT PPDAT50={VEL 100.000,ACC 100.000,APO_DIST 100.000,GEAR_JERK 50.0000,EXAX_IGN 3}
DECL E6POS XP66={X 1413.07727,Y -617.876160,Z 1470.88220,A 59.8442421,B 77.7953720,C 170.783493,S 2,T 42,E1 43.6475182,E2 179.999115,E3 180.003891,E4 0.0,E5 0.0,E6 0.0}
DECL FDAT FP66={TOOL_NO 1,BASE_NO 0,IPO_FRAME #BASE,POINT2[] " ",TQ_STATE FALSE}
DECL PDAT PPDAT51={VEL 100.000,ACC 100.000,APO_DIST 100.000,GEAR_JERK 50.0000,EXAX_IGN 3}
DECL ATBg_Start_T AS_WDAT33={JobModeId 1306102413,ParamSetId -1047099609,StartTime 0.0,PreFlowTime 0.0,Channel1 0.0,Channel2 2.00000,Channel3 0.0,Channel4 0.0,Channel5 0.0,Channel6 0.0,Channel7 0.0,Channel8 0.0,PurgeTime 0.0}
DECL ATBg_Weld_T AW_WDAT33={JobModeId -187662529,ParamSetId -430485013,Velocity 0.00830000,Channel1 30.0000,Channel2 1.00000,Channel3 0.0,Channel4 0.0,Channel5 0.0,Channel6 0.0,Channel7 0.0,Channel8 0.0}
DECL WTCg_WeaveDefinition_T WV_WDAT33={Pattern #None,Length 4.00000,Amplitude 2.00000,Angle 0.0}
DECL FDAT FP67={TOOL_NO 1,BASE_NO 0,IPO_FRAME #BASE,POINT2[] " ",TQ_STATE FALSE}
DECL PDAT PPDAT52={ACC 100.000,APO_DIST 100.000,APO_MODE #CPTP,GEAR_JERK 50.0000}
DECL E6POS XP67={X 1516.23657,Y -542.109131,Z 1407.86389,A 70.5701447,B 77.8772049,C 177.723236,S 2,T 42,E1 39.6729126,E2 179.999115,E3 180.003891,E4 0.0,E5 0.0,E6 0.0}
DECL ATBg_Crater_T AC_WDAT34={JobModeId -187662529,ParamSetId -1375177600,CraterTime 0.100000,PostflowTime 0.100000,Channel1 30.0000,Channel2 1.00000,Channel3 0.0,Channel4 0.0,Channel5 0.0,Channel6 0.0,Channel7 0.0,Channel8 0.0,BurnBackTime 0.0}
DECL FDAT FP68={TOOL_NO 1,BASE_NO 0,IPO_FRAME #BASE,POINT2[] " ",TQ_STATE FALSE}
DECL LDAT LCPDAT19={ACC 100.000,APO_DIST 100.000,APO_FAC 50.0000,AXIS_VEL 100.000,AXIS_ACC 100.000,ORI_TYP #VAR,CIRC_TYP #BASE,JERK_FAC 50.0000,GEAR_JERK 50.0000,EXAX_IGN 0}
DECL E6POS XP68={X 1516.23657,Y -542.109131,Z 1407.86389,A 70.5701447,B 77.8772049,C 177.723236,S 2,T 42,E1 39.6729126,E2 179.999115,E3 180.003891,E4 0.0,E5 0.0,E6 0.0}
DECL E6POS XP69={X 1382.02527,Y -494.258209,Z 1553.51624,A 50.0575943,B 77.0593185,C 156.721603,S 2,T 42,E1 39.6729126,E2 179.999115,E3 180.003891,E4 0.0,E5 0.0,E6 0.0}
DECL FDAT FP69={TOOL_NO 1,BASE_NO 0,IPO_FRAME #BASE,POINT2[] " ",TQ_STATE FALSE}
DECL PDAT PPDAT53={VEL 100.000,ACC 100.000,APO_DIST 100.000,GEAR_JERK 50.0000,EXAX_IGN 3}
DECL ATBg_Start_T AS_WDAT35={JobModeId 1306102413,ParamSetId -1047099609,StartTime 0.0,PreFlowTime 0.0,Channel1 0.0,Channel2 2.00000,Channel3 0.0,Channel4 0.0,Channel5 0.0,Channel6 0.0,Channel7 0.0,Channel8 0.0,PurgeTime 0.0}
DECL ATBg_Weld_T AW_WDAT35={JobModeId -187662529,ParamSetId -430485013,Velocity 0.00830000,Channel1 30.0000,Channel2 1.00000,Channel3 0.0,Channel4 0.0,Channel5 0.0,Channel6 0.0,Channel7 0.0,Channel8 0.0}
DECL WTCg_WeaveDefinition_T WV_WDAT35={Pattern #None,Length 4.00000,Amplitude 2.00000,Angle 0.0}
DECL FDAT FP70={TOOL_NO 1,BASE_NO 0,IPO_FRAME #BASE,POINT2[] " ",TQ_STATE FALSE}
DECL PDAT PPDAT54={ACC 100.000,APO_DIST 100.000,APO_MODE #CPTP,GEAR_JERK 50.0000}
DECL E6POS XP70={X 1579.26611,Y -136.946945,Z 1436.00012,A -88.2805939,B 58.3568497,C 3.02447629,S 2,T 10,E1 35.4823723,E2 180.095947,E3 180.003891,E4 0.0,E5 0.0,E6 0.0}
DECL ATBg_Crater_T AC_WDAT36={JobModeId -187662529,ParamSetId -1375177600,CraterTime 0.100000,PostflowTime 0.100000,Channel1 30.0000,Channel2 1.00000,Channel3 0.0,Channel4 0.0,Channel5 0.0,Channel6 0.0,Channel7 0.0,Channel8 0.0,BurnBackTime 0.0}
DECL FDAT FP71={TOOL_NO 1,BASE_NO 0,IPO_FRAME #BASE,POINT2[] " ",TQ_STATE FALSE}
DECL LDAT LCPDAT20={ACC 100.000,APO_DIST 100.000,APO_FAC 50.0000,AXIS_VEL 100.000,AXIS_ACC 100.000,ORI_TYP #VAR,CIRC_TYP #BASE,JERK_FAC 50.0000,GEAR_JERK 50.0000,EXAX_IGN 0}
DECL E6POS XP71={X 1579.26611,Y -136.946945,Z 1436.00012,A -88.2805939,B 58.3568497,C 3.02447629,S 2,T 10,E1 35.4823723,E2 180.095947,E3 180.003891,E4 0.0,E5 0.0,E6 0.0}
DECL E6POS XP72={X 1415.25378,Y -117.767067,Z 1567.15686,A -96.8179398,B 59.2228050,C -10.1517134,S 2,T 10,E1 35.4823723,E2 180.095947,E3 180.003891,E4 0.0,E5 0.0,E6 0.0}
DECL FDAT FP72={TOOL_NO 1,BASE_NO 0,IPO_FRAME #BASE,POINT2[] " ",TQ_STATE FALSE}
DECL PDAT PPDAT55={VEL 100.000,ACC 100.000,APO_DIST 100.000,GEAR_JERK 50.0000,EXAX_IGN 3}
DECL E6POS XP73={X 1415.25378,Y -117.767067,Z 1567.15686,A -96.8179398,B 59.2228050,C -10.1517162,S 2,T 10,E1 35.4823723,E2 180.095947,E3 180.003891,E4 0.0,E5 0.0,E6 0.0}
DECL FDAT FP73={TOOL_NO 1,BASE_NO 0,IPO_FRAME #BASE,POINT2[] " ",TQ_STATE FALSE}
DECL PDAT PPDAT56={VEL 100.000,ACC 100.000,APO_DIST 100.000,GEAR_JERK 50.0000,EXAX_IGN 3}
DECL ATBg_Start_T AS_WDAT37={JobModeId 1306102413,ParamSetId -1047099609,StartTime 0.0,PreFlowTime 0.0,Channel1 0.0,Channel2 2.00000,Channel3 0.0,Channel4 0.0,Channel5 0.0,Channel6 0.0,Channel7 0.0,Channel8 0.0,PurgeTime 0.0}
DECL ATBg_Weld_T AW_WDAT37={JobModeId -187662529,ParamSetId -430485013,Velocity 0.00830000,Channel1 30.0000,Channel2 1.00000,Channel3 0.0,Channel4 0.0,Channel5 0.0,Channel6 0.0,Channel7 0.0,Channel8 0.0}
DECL WTCg_WeaveDefinition_T WV_WDAT37={Pattern #None,Length 4.00000,Amplitude 2.00000,Angle 0.0}
DECL FDAT FP74={TOOL_NO 1,BASE_NO 0,IPO_FRAME #BASE,POINT2[] " ",TQ_STATE FALSE}
DECL PDAT PPDAT57={ACC 100.000,APO_DIST 100.000,APO_MODE #CPTP,GEAR_JERK 50.0000}
DECL E6POS XP74={X 1584.38623,Y 111.410187,Z 1386.96509,A 102.267334,B 52.8598785,C -171.791306,S 2,T 43,E1 30.6981010,E2 180.095947,E3 180.003891,E4 0.0,E5 0.0,E6 0.0}
DECL ATBg_Crater_T AC_WDAT38={JobModeId -187662529,ParamSetId -1375177600,CraterTime 0.100000,PostflowTime 0.100000,Channel1 30.0000,Channel2 1.00000,Channel3 0.0,Channel4 0.0,Channel5 0.0,Channel6 0.0,Channel7 0.0,Channel8 0.0,BurnBackTime 0.0}
DECL FDAT FP75={TOOL_NO 1,BASE_NO 0,IPO_FRAME #BASE,POINT2[] " ",TQ_STATE FALSE}
DECL LDAT LCPDAT21={ACC 100.000,APO_DIST 100.000,APO_FAC 50.0000,AXIS_VEL 100.000,AXIS_ACC 100.000,ORI_TYP #VAR,CIRC_TYP #BASE,JERK_FAC 50.0000,GEAR_JERK 50.0000,EXAX_IGN 0}
DECL E6POS XP75={X 1584.38623,Y 111.410187,Z 1386.96509,A 102.267334,B 52.8598785,C -171.791306,S 2,T 43,E1 30.6981010,E2 180.095947,E3 180.003891,E4 0.0,E5 0.0,E6 0.0}
DECL E6POS XP76={X 1441.27734,Y -90.4894485,Z 1536.43652,A -100.739212,B 68.4979858,C -14.1514530,S 2,T 10,E1 34.8087654,E2 180.095947,E3 180.003891,E4 0.0,E5 0.0,E6 0.0}
DECL FDAT FP76={TOOL_NO 1,BASE_NO 0,IPO_FRAME #BASE,POINT2[] " ",TQ_STATE FALSE}
DECL PDAT PPDAT58={VEL 100.000,ACC 100.000,APO_DIST 100.000,GEAR_JERK 50.0000,EXAX_IGN 3}
DECL E6POS XP77={X 1472.05359,Y -555.361511,Z 1447.94543,A 53.5533104,B 56.5259285,C 162.220825,S 2,T 42,E1 180.000992,E2 179.999115,E3 180.003891,E4 0.0,E5 0.0,E6 0.0}
DECL FDAT FP77={TOOL_NO 1,BASE_NO 0,IPO_FRAME #BASE,POINT2[] " ",TQ_STATE FALSE}
DECL PDAT PPDAT59={VEL 100.000,ACC 100.000,APO_DIST 100.000,GEAR_JERK 50.0000,EXAX_IGN 3}
DECL ATBg_Start_T AS_WDAT39={JobModeId 1306102413,ParamSetId -1047099609,StartTime 0.0,PreFlowTime 0.0,Channel1 0.0,Channel2 2.00000,Channel3 0.0,Channel4 0.0,Channel5 0.0,Channel6 0.0,Channel7 0.0,Channel8 0.0,PurgeTime 0.0}
DECL ATBg_Weld_T AW_WDAT39={JobModeId 1306102413,ParamSetId -540622874,Velocity 0.00830000,Channel1 0.0,Channel2 1.00000,Channel3 0.0,Channel4 0.0,Channel5 0.0,Channel6 0.0,Channel7 0.0,Channel8 0.0}
DECL WTCg_WeaveDefinition_T WV_WDAT39={Pattern #None,Length 4.00000,Amplitude 2.00000,Angle 0.0}
DECL FDAT FP78={TOOL_NO 1,BASE_NO 0,IPO_FRAME #BASE,POINT2[] " ",TQ_STATE FALSE}
DECL PDAT PPDAT60={ACC 100.000,APO_DIST 100.000,APO_MODE #CPTP,GEAR_JERK 50.0000}
DECL E6POS XP78={X 1344.34131,Y 545.107666,Z 1613.57458,A 101.826927,B 70.2007828,C 176.589447,S 2,T 35,E1 229.997406,E2 195.002228,E3 195.004227,E4 0.0,E5 0.0,E6 0.0}
DECL ATBg_Crater_T AC_WDAT40={JobModeId -187662529,ParamSetId -1375177600,CraterTime 0.100000,PostflowTime 0.100000,Channel1 30.0000,Channel2 1.00000,Channel3 0.0,Channel4 0.0,Channel5 0.0,Channel6 0.0,Channel7 0.0,Channel8 0.0,BurnBackTime 0.0}
DECL FDAT FP79={TOOL_NO 1,BASE_NO 0,IPO_FRAME #BASE,POINT2[] " ",TQ_STATE FALSE}
DECL LDAT LCPDAT22={ACC 100.000,APO_DIST 100.000,APO_FAC 50.0000,AXIS_VEL 100.000,AXIS_ACC 100.000,ORI_TYP #VAR,CIRC_TYP #BASE,JERK_FAC 50.0000,GEAR_JERK 50.0000,EXAX_IGN 0}
DECL E6POS XP79={X 1345.37646,Y 533.994629,Z 1613.35364,A 102.084946,B 70.2269897,C 176.990280,S 2,T 35,E1 229.997406,E2 195.002228,E3 195.004227,E4 0.0,E5 0.0,E6 0.0}
DECL ATBg_Start_T AS_WDAT41={JobModeId -187662529,ParamSetId 687014726,StartTime 0.0,PreFlowTime 0.100000,Channel1 30.0000,Channel2 1.00000,Channel3 0.0,Channel4 0.0,Channel5 0.0,Channel6 0.0,Channel7 0.0,Channel8 0.0,PurgeTime 0.0}
DECL ATBg_Weld_T AW_WDAT41={JobModeId -187662529,ParamSetId -430485013,Velocity 0.00830000,Channel1 30.0000,Channel2 1.00000,Channel3 0.0,Channel4 0.0,Channel5 0.0,Channel6 0.0,Channel7 0.0,Channel8 0.0}
DECL WTCg_WeaveDefinition_T WV_WDAT41={Pattern #None,Length 4.00000,Amplitude 2.00000,Angle 0.0}
DECL FDAT FP80={TOOL_NO 1,BASE_NO 0,IPO_FRAME #BASE,POINT2[] " ",TQ_STATE FALSE}
DECL PDAT PPDAT61={ACC 100.000,APO_DIST 100.000,APO_MODE #CPTP,GEAR_JERK 50.0000}
DECL E6POS XP80={X 1389.51404,Y 302.941376,Z 1610.34790,A 104.640984,B 74.7491074,C -177.070221,S 2,T 35,E1 229.997360,E2 195.002197,E3 195.004211,E4 0.0,E5 0.0,E6 0.0}
DECL ATBg_Crater_T AC_WDAT42={JobModeId -187662529,ParamSetId -1375177600,CraterTime 0.100000,PostflowTime 0.100000,Channel1 30.0000,Channel2 1.00000,Channel3 0.0,Channel4 0.0,Channel5 0.0,Channel6 0.0,Channel7 0.0,Channel8 0.0,BurnBackTime 0.0}
DECL FDAT FP81={TOOL_NO 1,BASE_NO 0,IPO_FRAME #BASE,POINT2[] " ",TQ_STATE FALSE}
DECL LDAT LCPDAT23={ACC 100.000,APO_DIST 100.000,APO_FAC 50.0000,AXIS_VEL 100.000,AXIS_ACC 100.000,ORI_TYP #VAR,CIRC_TYP #BASE,JERK_FAC 50.0000,GEAR_JERK 50.0000,EXAX_IGN 0}
DECL E6POS XP81={X 1391.36011,Y 294.178101,Z 1611.30188,A 106.205254,B 80.0392685,C -175.542023,S 2,T 35,E1 229.997360,E2 195.002197,E3 195.004211,E4 0.0,E5 0.0,E6 0.0}
DECL ATBg_Start_T AS_WDAT43={JobModeId -187662529,ParamSetId 687014726,StartTime 0.0,PreFlowTime 0.100000,Channel1 30.0000,Channel2 1.00000,Channel3 0.0,Channel4 0.0,Channel5 0.0,Channel6 0.0,Channel7 0.0,Channel8 0.0,PurgeTime 0.0}
DECL ATBg_Weld_T AW_WDAT43={JobModeId -187662529,ParamSetId -430485013,Velocity 0.00830000,Channel1 30.0000,Channel2 1.00000,Channel3 0.0,Channel4 0.0,Channel5 0.0,Channel6 0.0,Channel7 0.0,Channel8 0.0}
DECL WTCg_WeaveDefinition_T WV_WDAT43={Pattern #None,Length 4.00000,Amplitude 2.00000,Angle 0.0}
DECL FDAT FP82={TOOL_NO 1,BASE_NO 0,IPO_FRAME #BASE,POINT2[] " ",TQ_STATE FALSE}
DECL PDAT PPDAT62={ACC 100.000,APO_DIST 100.000,APO_MODE #CPTP,GEAR_JERK 50.0000}
DECL E6POS XP82={X 1405.05640,Y -51.4842529,Z 1609.80847,A 140.270340,B 86.4778442,C -127.943268,S 2,T 34,E1 229.997360,E2 195.002197,E3 195.004211,E4 0.0,E5 0.0,E6 0.0}
DECL ATBg_Crater_T AC_WDAT44={JobModeId -187662529,ParamSetId -1375177600,CraterTime 0.100000,PostflowTime 0.100000,Channel1 30.0000,Channel2 1.00000,Channel3 0.0,Channel4 0.0,Channel5 0.0,Channel6 0.0,Channel7 0.0,Channel8 0.0,BurnBackTime 0.0}
DECL FDAT FP83={TOOL_NO 1,BASE_NO 0,IPO_FRAME #BASE,POINT2[] " ",TQ_STATE FALSE}
DECL LDAT LCPDAT24={ACC 100.000,APO_DIST 100.000,APO_FAC 50.0000,AXIS_VEL 100.000,AXIS_ACC 100.000,ORI_TYP #VAR,CIRC_TYP #BASE,JERK_FAC 50.0000,GEAR_JERK 50.0000,EXAX_IGN 0}
DECL E6POS XP83={X 1405.05640,Y -51.4842529,Z 1609.80847,A 140.270340,B 86.4778442,C -127.943268,S 2,T 34,E1 229.997360,E2 195.002197,E3 195.004211,E4 0.0,E5 0.0,E6 0.0}
DECL E6POS XP84={X 1399.90735,Y -51.4098587,Z 1616.55884,A 136.356430,B 86.7458420,C -131.864014,S 2,T 34,E1 229.997360,E2 195.002197,E3 195.004211,E4 0.0,E5 0.0,E6 0.0}
DECL FDAT FP84={TOOL_NO 1,BASE_NO 0,IPO_FRAME #BASE,POINT2[] " ",TQ_STATE FALSE}
DECL PDAT PPDAT63={VEL 100.000,ACC 100.000,APO_DIST 100.000,APO_MODE #CDIS,GEAR_JERK 50.0000,EXAX_IGN 3}
DECL E6POS XP85={X 1319.20300,Y -50.2438545,Z 1728.13440,A 26.8801632,B 85.2404327,C 118.532234,S 2,T 34,E1 229.997360,E2 195.002197,E3 195.004211,E4 0.0,E5 0.0,E6 0.0}
DECL FDAT FP85={TOOL_NO 1,BASE_NO 0,IPO_FRAME #BASE,POINT2[] " ",TQ_STATE FALSE}
DECL PDAT PPDAT64={VEL 100.000,ACC 100.000,APO_DIST 100.000,APO_MODE #CDIS,GEAR_JERK 50.0000,EXAX_IGN 3}
DECL E6POS XP86={X 1308.38721,Y -175.908188,Z 1728.13440,A 21.4040012,B 85.2404327,C 118.532234,S 2,T 34,E1 229.997360,E2 195.002197,E3 195.004211,E4 0.0,E5 0.0,E6 0.0}
DECL FDAT FP86={TOOL_NO 1,BASE_NO 0,IPO_FRAME #BASE,POINT2[] " ",TQ_STATE FALSE}
DECL PDAT PPDAT65={VEL 100.000,ACC 100.000,APO_DIST 100.000,APO_MODE #CDIS,GEAR_JERK 50.0000,EXAX_IGN 3}
DECL ATBg_Start_T AS_WDAT45={JobModeId -187662529,ParamSetId 687014726,StartTime 0.0,PreFlowTime 0.100000,Channel1 30.0000,Channel2 1.00000,Channel3 0.0,Channel4 0.0,Channel5 0.0,Channel6 0.0,Channel7 0.0,Channel8 0.0,PurgeTime 0.0}
DECL ATBg_Weld_T AW_WDAT45={JobModeId -187662529,ParamSetId -430485013,Velocity 0.00830000,Channel1 30.0000,Channel2 1.00000,Channel3 0.0,Channel4 0.0,Channel5 0.0,Channel6 0.0,Channel7 0.0,Channel8 0.0}
DECL WTCg_WeaveDefinition_T WV_WDAT45={Pattern #None,Length 4.00000,Amplitude 2.00000,Angle 0.0}
